// TwinCAT 3 PLC project TcDynCollectionsTest
// Title: TwinCAT Dynamic Collections Test
// Company: FisoThemes
// Author: Goodwill Mzumala
// Description: Test solution for the TcDynCollections Library
// ProgramVersion: 3.1.4023.0
// libraries:
//   Tc2_Standard, * (Beckhoff Automation GmbH)
//   Tc2_System, * (Beckhoff Automation GmbH)
//   Tc2_Utilities, * (Beckhoff Automation GmbH)
//   Tc3_Module, * (Beckhoff Automation GmbH)
//   TcUnit, * (www.tcunit.org)
//   TwinCat Dynamic Collections, * (FisoThemes)
// project tree:
//   / PlcTask.TcTTO
//   POUs/Function Blocks/ FB_Array_List_Test_Suite.TcPOU, FB_Array_Test_Suite.TcPOU, FB_Ordered_Hash_Map_Test_Suite.TcPOU, FB_Ordered_Hash_Set_Test_Suite.TcPOU, FB_List_Test_Suite.TcPOU, FB_Queue_Test_Suite.TcPOU, FB_Deque_Test_Suite.TcPOU, FB_Stack_Test_Suite.TcPOU, FB_Tree_Map_Test_Suite.TcPOU, FB_Hash_Map_Test_Suite.TcPOU, FB_Tree_Set_Test_Suite.TcPOU, FB_Tree_Multiset_Test_Suite.TcPOU, FB_Hash_Set_Test_Suite.TcPOU
//   POUs/ MAIN.TcPOU
// (motion and I/O tree: see PLC project tcdyncollections)
// real-time tasks:
//   TASK PlcTask: cycle T#10ms, priority 20, ADS port 350
//   TASK PlcTestTask: cycle T#10ms, priority 21, ADS port 353

CONFIGURATION TcDynCollectionsTest
    RESOURCE PLC ON TwinCAT3
        TASK PlcTask(INTERVAL := T#10ms, PRIORITY := 20);
        PROGRAM MAIN WITH PlcTask : MAIN;
    END_RESOURCE
END_CONFIGURATION

// ---- POUs/MAIN.TcPOU
PROGRAM MAIN
VAR
	fbArray_List_Test_Suite : FB_Array_List_Test_Suite;
	fbList_Test_Suite : FB_List_Test_Suite;
	fbArray_Test_Suite : FB_Array_Test_Suite;
	fbQueue_Test_Suite : FB_Queue_Test_Suite;
	fbStack_Test_Suite : FB_Stack_Test_Suite;
	fbDeque_Test_Suite : FB_Deque_Test_Suite;
	fbTree_Set_Test_Suite : FB_Tree_Set_Test_Suite;
	fbTree_Map_Test_Suite : FB_Tree_Map_Test_Suite;
	fbTree_Multiset_Test_Suite : FB_Tree_Multiset_Test_Suite;
	fbHash_Set_Test_Suite : FB_Hash_Set_Test_Suite;
	fbHash_Map_Test_Suite : FB_Hash_Map_Test_Suite;
	fbOrdered_Hash_Set_Test_Suite : FB_Ordered_Hash_Set_Test_Suite;
	fbOrdered_Hash_Map_Test_Suite : FB_Ordered_Hash_Map_Test_Suite;
END_VAR

TcUnit.RUN();

END_PROGRAM

// ---- POUs/Function Blocks/FB_Array_List_Test_Suite.TcPOU
FUNCTION_BLOCK FB_Array_List_Test_Suite EXTENDS TcUnit.FB_TestSuite
VAR
END_VAR

THIS^.Append_Items_And_Check_If_Count_Changes();
THIS^.Append_Items_And_Get_Items();
THIS^.Prepend_Items_And_Get_Items();
THIS^.Append_Items_Reverse_The_List_And_Get_Items();
THIS^.Append_Find_Item_Indices_And_Get_Items_With_Them();
THIS^.Remove_Tests();
THIS^.Set_Value_At_Index_To_Item_And_Get_Item();

// Test appending multiple elements, finds them and verify values using the get method.
METHOD Append_Find_Item_Indices_And_Get_Items_With_Them
VAR_INST
	fbList 		: TcDynCollections.FB_Array_List(0);
	Idx 		: ARRAY[0..4] OF TcDynCollections.T_Position;
	arbValue 	: ARRAY[0..2] OF BOOL := [TRUE, TRUE];
	arnValue 	: ARRAY[0..2] OF INT := [33, 33];
	arsValue 	: ARRAY[0..2] OF STRING := ['I love cats.', 'I love cats.'];
	arwsValue 	: ARRAY[0..2] OF WSTRING := ["I love dogs.", "I love dogs."];
	arfValue 	: ARRAY[0..2] OF LREAL := [21.3, 21.3];
END_VAR
TcUnit.TEST('Append_Find_Item_Indices_And_Get_Items_With_Them');

	fbList
		.Append(arbValue[0])
		.Append(arnValue[0])
		.Append(arsValue[0])
		.Append(arwsValue[0])
		.Append(arfValue[0]);

	// Make the strings dirty. 	
	arsValue[0] 	:= 'kjhsadkfjvhbkjhdfbkvsjhbfkvjhsbkfv';
	arwsValue[0] 	:= "kjhsadkfjvhbkjhdfbkvsjhbfkvjhsbkfv";
	arsValue[0] 	:= 'I love cats.';
	arwsValue[0] 	:= "I love dogs.";
		
	fbList
		.Search(arbValue[0], Index => Idx[0])
		.Search(arnValue[0], Index => Idx[1])
		.Search(arsValue[0], Index => Idx[2])
		.Search(arwsValue[0],Index => Idx[3])
		.Search(arfValue[0], Index => Idx[4]);
		
	fbList
		.Get(Idx[0], arbValue[2])
		.Get(Idx[1], arnValue[2])
		.Get(Idx[2], arsValue[2])
		.Get(Idx[3], arwsValue[2])
		.Get(Idx[4], arfValue[2]);
		
	THIS^.AssertEquals_DINT(5, fbList._Count, 'List item count must be 5 after after appending items to list.');
	THIS^.AssertEquals_BOOL(arbValue[1], arbValue[2], 'Appended BOOL item is not what is expected after the get operation.');
	THIS^.AssertEquals_INT(arnValue[1], arnValue[2], 'Appended INT item is not what is expected after the get operation.');
	THIS^.AssertEquals_STRING(arsValue[1], arsValue[2], 'Appended STRING item is not what is expected after the get operation.');
	THIS^.AssertEquals_WSTRING(arwsValue[1], arwsValue[2], 'Appended STRING item is not what is expected after the get operation.');
	THIS^.AssertEquals_LREAL(arfValue[1], arfValue[2],0.01, 'Appended LREAL item is not what is expected after the get operation.');

	TEST_FINISHED();
END_METHOD

// 1) Test that a newly created FB_Array_List has an item count of 0 and is empty.
// 2) Test that after appending elements, the size increases accordingly and is no longer empty.
// 3) Test that after removing all elements, the size becomes 0 again and the list is empty.
METHOD Append_Items_And_Check_If_Count_Changes
VAR_INST
	fbList : TcDynCollections.FB_Array_List(0);
	nValue : INT := 33;
	sValue : STRING := 'I love cats.';
END_VAR
TcUnit.TEST('Append_Items_And_Check_If_Count_Changes');

	THIS^.AssertEquals_DINT(0, fbList._Count, 'List item count must be 0.');
	THIS^.AssertEquals_BOOL(TRUE, fbList._Empty, '_Empty property didnt return TRUE.');
	
	fbList
		.Append(nValue)
		.Append(sValue);
	
	THIS^.AssertEquals_DINT(2, fbList._Count, 'List item count must be 2 after appending values.');
	THIS^.AssertEquals_BOOL(FALSE, fbList._Empty, '_Empty property didnt return FALSE after appending value.');
	
	fbList.Clear();
	
	THIS^.AssertEquals_DINT(0, fbList._Count, 'List item count must be 0 after clearing list.');
	THIS^.AssertEquals_BOOL(TRUE, fbList._Empty, '_Empty property didnt return TRUE after clearing list.');
	
	TEST_FINISHED();
END_METHOD

// Test appending multiple elements and verify their order and values using the get method.
METHOD Append_Items_And_Get_Items
VAR_INST
	fbList 		: TcDynCollections.FB_Array_List(0);
	
	arbValue 	: ARRAY[0..2] OF BOOL := [TRUE, TRUE];
	arnValue 	: ARRAY[0..2] OF INT := [33, 33];
	arsValue 	: ARRAY[0..2] OF STRING := ['I love cats.', 'I love cats.'];
	arwsValue 	: ARRAY[0..2] OF WSTRING := ["I love dogs.", "I love dogs."];
	arfValue 	: ARRAY[0..2] OF LREAL := [21.3, 21.3];
END_VAR
TcUnit.TEST('Append_Items_And_Get_Items');

	fbList
		.Append(arbValue[0])
		.Append(arnValue[0])
		.Append(arsValue[0])
		.Append(arwsValue[0])
		.Append(arfValue[0]);
		
	fbList
		.Get(0, arbValue[2])
		.Get(1, arnValue[2])
		.Get(2, arsValue[2])
		.Get(3, arwsValue[2])
		.Get(4, arfValue[2]);
		
	THIS^.AssertEquals_DINT(5, fbList._Count, 'List item count must be 5 after after appending items to list.');
	THIS^.AssertEquals_BOOL(arbValue[1], arbValue[2], 'Appended BOOL item is not what is expected after the get operation.');
	THIS^.AssertEquals_INT(arnValue[1], arnValue[2], 'Appended INT item is not what is expected after the get operation.');
	THIS^.AssertEquals_STRING(arsValue[1], arsValue[2], 'Appended STRING item is not what is expected after the get operation.');
	THIS^.AssertEquals_WSTRING(arwsValue[1], arwsValue[2], 'Appended STRING item is not what is expected after the get operation.');
	THIS^.AssertEquals_LREAL(arfValue[1], arfValue[2],0.01, 'Appended LREAL item is not what is expected after the get operation.');

	TEST_FINISHED();
END_METHOD

// Test appending multiple elements, reversing their order and verifiying their order and values using the get method.
METHOD Append_Items_Reverse_The_List_And_Get_Items
VAR_INST
	fbList 		: TcDynCollections.FB_Array_List(0);
	
	arbValue 	: ARRAY[0..2] OF BOOL := [TRUE, TRUE];
	arnValue 	: ARRAY[0..2] OF INT := [33, 33];
	arsValue 	: ARRAY[0..2] OF STRING := ['I love cats.', 'I love cats.'];
	arwsValue 	: ARRAY[0..2] OF WSTRING := ["I love dogs.", "I love dogs."];
	arfValue 	: ARRAY[0..2] OF LREAL := [21.3, 21.3];
END_VAR
TcUnit.TEST('Append_Items_Reverse_The_List_And_Get_Items');

	fbList
		.Append(arbValue[0])
		.Append(arnValue[0])
		.Append(arsValue[0])
		.Append(arwsValue[0])
		.Append(arfValue[0])
		.Reverse();
		
	fbList
		.Get(4, arbValue[2])
		.Get(3, arnValue[2])
		.Get(2, arsValue[2])
		.Get(1, arwsValue[2])
		.Get(0, arfValue[2]);
		
	THIS^.AssertEquals_DINT(5, fbList._Count, 'List item count must be 5 after after appending items to list.');
	THIS^.AssertEquals_BOOL(arbValue[1], arbValue[2], 'Appended BOOL item is not what is expected after the get operation.');
	THIS^.AssertEquals_INT(arnValue[1], arnValue[2], 'Appended INT item is not what is expected after the get operation.');
	THIS^.AssertEquals_STRING(arsValue[1], arsValue[2], 'Appended STRING item is not what is expected after the get operation.');
	THIS^.AssertEquals_WSTRING(arwsValue[1], arwsValue[2], 'Appended STRING item is not what is expected after the get operation.');
	THIS^.AssertEquals_LREAL(arfValue[1], arfValue[2],0.01, 'Appended LREAL item is not what is expected after the get operation.');

	TEST_FINISHED();
END_METHOD

// Test prepending multiple elements and verify their order and values using the get method.
METHOD Prepend_Items_And_Get_Items
VAR_INST
	fbList 		: TcDynCollections.FB_Array_List(0);
	
	arbValue 	: ARRAY[0..2] OF BOOL := [TRUE, TRUE];
	arnValue 	: ARRAY[0..2] OF INT := [33, 33];
	arsValue 	: ARRAY[0..2] OF STRING := ['I love cats.', 'I love cats.'];
	arwsValue 	: ARRAY[0..2] OF WSTRING := ["I love dogs.", "I love dogs."];
	arfValue 	: ARRAY[0..2] OF LREAL := [21.3, 21.3];
END_VAR
TcUnit.TEST('Prepend_Items_And_Get_Items');

	fbList
		.Prepend(arbValue[0])
		.Prepend(arnValue[0])
		.Prepend(arsValue[0])
		.Prepend(arwsValue[0])
		.Prepend(arfValue[0]);
		
	fbList
		.Get(4, arbValue[2])
		.Get(3, arnValue[2])
		.Get(2, arsValue[2])
		.Get(1, arwsValue[2])
		.Get(0, arfValue[2]);
		
	THIS^.AssertEquals_DINT(5, fbList._Count, 'List item count must be 5 after after appending items to list.');
	THIS^.AssertEquals_BOOL(arbValue[1], arbValue[2], 'Appended BOOL item is not what is expected after the get operation.');
	THIS^.AssertEquals_INT(arnValue[1], arnValue[2], 'Appended INT item is not what is expected after the get operation.');
	THIS^.AssertEquals_STRING(arsValue[1], arsValue[2], 'Appended STRING item is not what is expected after the get operation.');
	THIS^.AssertEquals_WSTRING(arwsValue[1], arwsValue[2], 'Appended STRING item is not what is expected after the get operation.');
	THIS^.AssertEquals_LREAL(arfValue[1], arfValue[2],0.01, 'Appended LREAL item is not what is expected after the get operation.');

	TEST_FINISHED();
END_METHOD

// Test appending multiple elements, removing first item, verifying the size and values.
// 
METHOD Remove_Tests
VAR_INST
	fbList 		: TcDynCollections.FB_Array_List(0);
	i 			: TcDynCollections.T_Position;
	n 			: TcDynCollections.T_Capacity;
	arbValue 	: ARRAY[0..2] OF BOOL := [TRUE, TRUE];
	arnValue 	: ARRAY[0..2] OF INT := [33, 33];
	arsValue 	: ARRAY[0..2] OF STRING := ['I love cats.', 'I love cats.'];
	arwsValue 	: ARRAY[0..2] OF WSTRING := ["I love dogs.", "I love dogs."];
	arfValue 	: ARRAY[0..2] OF LREAL := [21.3, 21.3];
END_VAR
TcUnit.TEST('Remove_Tests');

	fbList
		.Append(arbValue[0])
		.Append(arnValue[0])
		.Append(arsValue[0])
		.Append(arwsValue[0])
		.Append(arfValue[0]);
		
	fbList
		.Remove(arbValue[0])
		.Get(0, arnValue[2]);
		
	THIS^.AssertEquals_DINT(4, fbList._Count, 'List item count must be 4 after appending and removing fisrt item at from the list.');
	THIS^.AssertEquals_INT(arnValue[1], arnValue[2],'');
	
	fbList
		.Prepend(arbValue[0])
		.Remove_At(2)
		.Get(2, arwsValue[2]);
		
	THIS^.AssertEquals_DINT(4, fbList._Count, 'List item count must be 4 after prepending removed item and removing item in index 2 of the list.');
	THIS^.AssertEquals_WSTRING(arwsValue[1], arwsValue[2], '');
	
	fbList
		.Insert(2, arsValue[0])
		.Remove_Last()
		.Get(3, arwsValue[2]);
		
	THIS^.AssertEquals_DINT(4, fbList._Count, 'List item count must be 4 after inserting removed from index 2 item and removing the last item in the list.');
	THIS^.AssertEquals_WSTRING(arwsValue[1], arwsValue[2], '');
	
	n := fbList._Count;
	FOR i := 0 TO n - 1 DO
		fbList.Remove_Last();
		END_FOR
		
	THIS^.AssertEquals_DINT(0, fbList._Count, 'List item count must be zero after removing all items from the back.');
	THIS^.AssertEquals_BOOL(TRUE, fbList._Empty, 'List _Empty property must be zero TRUE removing all items from the back.');
	
	FOR i := 0 TO 4 DO fbList.Prepend(arwsValue); END_FOR
	
	THIS^.AssertEquals_DINT(5, fbList._Count, 'Failed to prepend items to list for checking removing all items from the front.');
	
	n := fbList._Count;
	FOR i := 0 TO n - 1 DO
		fbList.Remove_At(0);
		END_FOR
		
	THIS^.AssertEquals_DINT(0, fbList._Count, 'List item count must be zero after removing all items from the front.');
	THIS^.AssertEquals_BOOL(TRUE, fbList._Empty, 'List _Empty property must be zero TRUE removing all items from the front.');

	TEST_FINISHED();
END_METHOD

// Test appending multiple elements and verify their order and values using the get method.
METHOD Set_Value_At_Index_To_Item_And_Get_Item
VAR_INST
	fbList 		: TcDynCollections.FB_Array_List(5);
	
	arbValue 	: ARRAY[0..2] OF BOOL := [TRUE, TRUE];
	arnValue 	: ARRAY[0..2] OF INT := [33, 33];
	arsValue 	: ARRAY[0..2] OF STRING := ['I love cats.', 'I love cats.'];
	arwsValue 	: ARRAY[0..2] OF WSTRING := ["I love dogs.", "I love dogs."];
	arfValue 	: ARRAY[0..2] OF LREAL := [21.3, 21.3];
END_VAR
TcUnit.TEST('Set_Value_At_Index_To_Item_And_Get_Item');

	fbList
		.Set(0, arbValue[0])
		.Set(1, arnValue[0])
		.Set(2, arsValue[0])
		.Set(3, arwsValue[0])
		.Set(4, arfValue[0]);
		
	fbList
		.Get(0, arbValue[2])
		.Get(1, arnValue[2])
		.Get(2, arsValue[2])
		.Get(3, arwsValue[2])
		.Get(4, arfValue[2]);
		
	THIS^.AssertEquals_DINT(5, fbList._Count, 'List item count must be 5 after after appending items to list.');
	THIS^.AssertEquals_BOOL(arbValue[1], arbValue[2], 'Appended BOOL item is not what is expected after the get operation.');
	THIS^.AssertEquals_INT(arnValue[1], arnValue[2], 'Appended INT item is not what is expected after the get operation.');
	THIS^.AssertEquals_STRING(arsValue[1], arsValue[2], 'Appended STRING item is not what is expected after the get operation.');
	THIS^.AssertEquals_WSTRING(arwsValue[1], arwsValue[2], 'Appended STRING item is not what is expected after the get operation.');
	THIS^.AssertEquals_LREAL(arfValue[1], arfValue[2],0.01, 'Appended LREAL item is not what is expected after the get operation.');

	TEST_FINISHED();
END_METHOD

END_FUNCTION_BLOCK

// ---- POUs/Function Blocks/FB_List_Test_Suite.TcPOU
FUNCTION_BLOCK FB_List_Test_Suite EXTENDS TcUnit.FB_TestSuite
VAR
END_VAR

THIS^.Append_Items_And_Check_If_Count_Changes();
THIS^.Append_Items_And_Get_Items();
THIS^.Prepend_Items_And_Get_Items();
THIS^.Append_Items_Reverse_The_List_And_Get_Items();
THIS^.Append_Find_Item_Indices_And_Get_Items_With_Them();
THIS^.Remove_Tests();
THIS^.Set_Value_At_Index_To_Item_And_Get_Item();

// Test appending multiple elements, finds them and verify values using the get method.
METHOD Append_Find_Item_Indices_And_Get_Items_With_Them
VAR_INST
	fbList 		: TcDynCollections.FB_List;
	Idx 		: ARRAY[0..4] OF TcDynCollections.T_Position;
	arbValue 	: ARRAY[0..2] OF BOOL := [TRUE, TRUE];
	arnValue 	: ARRAY[0..2] OF INT := [33, 33];
	arsValue 	: ARRAY[0..2] OF STRING := ['I love cats.', 'I love cats.'];
	arwsValue 	: ARRAY[0..2] OF WSTRING := ["I love dogs.", "I love dogs."];
	arfValue 	: ARRAY[0..2] OF LREAL := [21.3, 21.3];
END_VAR
TcUnit.TEST('Append_Find_Item_Indices_And_Get_Items_With_Them');

	fbList
		.Append(arbValue[0])
		.Append(arnValue[0])
		.Append(arsValue[0])
		.Append(arwsValue[0])
		.Append(arfValue[0]);

	// Make the strings dirty. 	
	arsValue[0] 	:= 'kjhsadkfjvhbkjhdfbkvsjhbfkvjhsbkfv';
	arwsValue[0] 	:= "kjhsadkfjvhbkjhdfbkvsjhbfkvjhsbkfv";
	arsValue[0] 	:= 'I love cats.';
	arwsValue[0] 	:= "I love dogs.";
		
	fbList
		.Search(arbValue[0], Index => Idx[0])
		.Search(arnValue[0], Index => Idx[1])
		.Search(arsValue[0], Index => Idx[2])
		.Search(arwsValue[0],Index => Idx[3])
		.Search(arfValue[0], Index => Idx[4]);
		
	fbList
		.Get(Idx[0], arbValue[2])
		.Get(Idx[1], arnValue[2])
		.Get(Idx[2], arsValue[2])
		.Get(Idx[3], arwsValue[2])
		.Get(Idx[4], arfValue[2]);
		
	THIS^.AssertEquals_DINT(5, fbList._Count, 'List item count must be 5 after after appending items to list.');
	THIS^.AssertEquals_BOOL(arbValue[1], arbValue[2], 'Appended BOOL item is not what is expected after the get operation.');
	THIS^.AssertEquals_INT(arnValue[1], arnValue[2], 'Appended INT item is not what is expected after the get operation.');
	THIS^.AssertEquals_STRING(arsValue[1], arsValue[2], 'Appended STRING item is not what is expected after the get operation.');
	THIS^.AssertEquals_WSTRING(arwsValue[1], arwsValue[2], 'Appended STRING item is not what is expected after the get operation.');
	THIS^.AssertEquals_LREAL(arfValue[1], arfValue[2],0.01, 'Appended LREAL item is not what is expected after the get operation.');

	TEST_FINISHED();
END_METHOD

// 1) Test that a newly created FB_Array_List has an item count of 0 and is empty.
// 2) Test that after appending elements, the size increases accordingly and is no longer empty.
// 3) Test that after removing all elements, the size becomes 0 again and the list is empty.
METHOD Append_Items_And_Check_If_Count_Changes
VAR_INST
	fbList : TcDynCollections.FB_List;
	nValue : INT := 33;
	sValue : STRING := 'I love cats.';
END_VAR
TcUnit.TEST('Append_Items_And_Check_If_Count_Changes');

	THIS^.AssertEquals_DINT(0, fbList._Count, 'List item count must be 0.');
	THIS^.AssertEquals_BOOL(TRUE, fbList._Empty, 'Is_Empty property didnt return TRUE.');
	
	fbList
		.Append(nValue)
		.Append(sValue);
	
	THIS^.AssertEquals_DINT(2, fbList._Count, 'List item count must be 2 after appending values.');
	THIS^.AssertEquals_BOOL(FALSE, fbList._Empty, 'Is_Empty property didnt return FALSE after appending value.');
	
	fbList.Clear();
	
	THIS^.AssertEquals_DINT(0, fbList._Count, 'List item count must be 0 after clearing list.');
	THIS^.AssertEquals_BOOL(TRUE, fbList._Empty, 'Is_Empty property didnt return TRUE after clearing list.');
	
	TEST_FINISHED();
END_METHOD

// Test appending multiple elements and verify their order and values using the get method.
METHOD Append_Items_And_Get_Items
VAR_INST
	fbList 		: TcDynCollections.FB_List;
	
	arbValue 	: ARRAY[0..2] OF BOOL := [TRUE, TRUE];
	arnValue 	: ARRAY[0..2] OF INT := [33, 33];
	arsValue 	: ARRAY[0..2] OF STRING := ['I love cats.', 'I love cats.'];
	arwsValue 	: ARRAY[0..2] OF WSTRING := ["I love dogs.", "I love dogs."];
	arfValue 	: ARRAY[0..2] OF LREAL := [21.3, 21.3];
END_VAR
TcUnit.TEST('Append_Items_And_Get_Items');

	fbList
		.Append(arbValue[0])
		.Append(arnValue[0])
		.Append(arsValue[0])
		.Append(arwsValue[0])
		.Append(arfValue[0]);
		
	fbList
		.Get(0, arbValue[2])
		.Get(1, arnValue[2])
		.Get(2, arsValue[2])
		.Get(3, arwsValue[2])
		.Get(4, arfValue[2]);
		
	THIS^.AssertEquals_DINT(5, fbList._Count, 'List item count must be 5 after after appending items to list.');
	THIS^.AssertEquals_BOOL(arbValue[1], arbValue[2], 'Appended BOOL item is not what is expected after the get operation.');
	THIS^.AssertEquals_INT(arnValue[1], arnValue[2], 'Appended INT item is not what is expected after the get operation.');
	THIS^.AssertEquals_STRING(arsValue[1], arsValue[2], 'Appended STRING item is not what is expected after the get operation.');
	THIS^.AssertEquals_WSTRING(arwsValue[1], arwsValue[2], 'Appended STRING item is not what is expected after the get operation.');
	THIS^.AssertEquals_LREAL(arfValue[1], arfValue[2],0.01, 'Appended LREAL item is not what is expected after the get operation.');

	TEST_FINISHED();
END_METHOD

// Test appending multiple elements, reversing their order and verifiying their order and values using the get method.
METHOD Append_Items_Reverse_The_List_And_Get_Items
VAR_INST
	fbList 		: TcDynCollections.FB_List;
	
	arbValue 	: ARRAY[0..2] OF BOOL := [TRUE, TRUE];
	arnValue 	: ARRAY[0..2] OF INT := [33, 33];
	arsValue 	: ARRAY[0..2] OF STRING := ['I love cats.', 'I love cats.'];
	arwsValue 	: ARRAY[0..2] OF WSTRING := ["I love dogs.", "I love dogs."];
	arfValue 	: ARRAY[0..2] OF LREAL := [21.3, 21.3];
END_VAR
TcUnit.TEST('Append_Items_Reverse_The_List_And_Get_Items');

	fbList
		.Append(arbValue[0])
		.Append(arnValue[0])
		.Append(arsValue[0])
		.Append(arwsValue[0])
		.Append(arfValue[0])
		.Reverse();
		
	fbList
		.Get(4, arbValue[2])
		.Get(3, arnValue[2])
		.Get(2, arsValue[2])
		.Get(1, arwsValue[2])
		.Get(0, arfValue[2]);
		
	THIS^.AssertEquals_DINT(5, fbList._Count, 'List item count must be 5 after after appending items to list.');
	THIS^.AssertEquals_BOOL(arbValue[1], arbValue[2], 'Appended BOOL item is not what is expected after the get operation.');
	THIS^.AssertEquals_INT(arnValue[1], arnValue[2], 'Appended INT item is not what is expected after the get operation.');
	THIS^.AssertEquals_STRING(arsValue[1], arsValue[2], 'Appended STRING item is not what is expected after the get operation.');
	THIS^.AssertEquals_WSTRING(arwsValue[1], arwsValue[2], 'Appended STRING item is not what is expected after the get operation.');
	THIS^.AssertEquals_LREAL(arfValue[1], arfValue[2],0.01, 'Appended LREAL item is not what is expected after the get operation.');

	TEST_FINISHED();
END_METHOD

// Test prepending multiple elements and verify their order and values using the get method.
METHOD Prepend_Items_And_Get_Items
VAR_INST
	fbList 		: TcDynCollections.FB_List;
	arsPrint 	: ARRAY[0..4] OF STRING;
	arbValue 	: ARRAY[0..2] OF BOOL := [TRUE, TRUE];
	arnValue 	: ARRAY[0..2] OF INT := [33, 33];
	arsValue 	: ARRAY[0..2] OF STRING := ['I love cats.', 'I love cats.'];
	arwsValue 	: ARRAY[0..2] OF WSTRING := ["I love dogs.", "I love dogs."];
	arfValue 	: ARRAY[0..2] OF LREAL := [21.3, 21.3];
END_VAR
TcUnit.TEST('Prepend_Items_And_Get_Items');

	fbList
		.Prepend(arbValue[0])
		.Prepend(arnValue[0])
		.Prepend(arsValue[0])
		.Prepend(arwsValue[0])
		.Prepend(arfValue[0]);
		
	fbList
		.Get(4, arbValue[2])
		.Get(3, arnValue[2])
		.Get(2, arsValue[2])
		.Get(1, arwsValue[2])
		.Get(0, arfValue[2]);
		
	THIS^.AssertEquals_DINT(5, fbList._Count, 'List item count must be 5 after after appending items to list.');
	THIS^.AssertEquals_BOOL(arbValue[1], arbValue[2], 'Appended BOOL item is not what is expected after the get operation.');
	THIS^.AssertEquals_INT(arnValue[1], arnValue[2], 'Appended INT item is not what is expected after the get operation.');
	THIS^.AssertEquals_STRING(arsValue[1], arsValue[2], 'Appended STRING item is not what is expected after the get operation.');
	THIS^.AssertEquals_WSTRING(arwsValue[1], arwsValue[2], 'Appended STRING item is not what is expected after the get operation.');
	THIS^.AssertEquals_LREAL(arfValue[1], arfValue[2],0.01, 'Appended LREAL item is not what is expected after the get operation.');

	TEST_FINISHED();
END_METHOD

// Test appending multiple elements, removing first item, verifying the size and values.
METHOD Remove_Tests
VAR_INST
	fbList 		: TcDynCollections.FB_List;
	i 			: TcDynCollections.T_Position;
	n 			: TcDynCollections.T_Capacity;
	arbValue 	: ARRAY[0..2] OF BOOL := [TRUE, TRUE];
	arnValue 	: ARRAY[0..2] OF INT := [33, 33];
	arsValue 	: ARRAY[0..2] OF STRING := ['I love cats.', 'I love cats.'];
	arwsValue 	: ARRAY[0..2] OF WSTRING := ["I love dogs.", "I love dogs."];
	arfValue 	: ARRAY[0..2] OF LREAL := [21.3, 21.3];
END_VAR
TcUnit.TEST('Remove_Tests');

	fbList
		.Append(arbValue[0])
		.Append(arnValue[0])
		.Append(arsValue[0])
		.Append(arwsValue[0])
		.Append(arfValue[0]);
		
	fbList
		.Remove(arbValue[0])
		.Get(0, arnValue[2]);
		
	THIS^.AssertEquals_DINT(4, fbList._Count, 'List item count must be 4 after appending and removing fisrt item at from the list.');
	THIS^.AssertEquals_INT(arnValue[1], arnValue[2],'');
	
	fbList
		.Prepend(arbValue[0])
		.Remove_At(2)
		.Get(2, arwsValue[2]);
		
	THIS^.AssertEquals_DINT(4, fbList._Count, 'List item count must be 4 after prepending removed item and removing item in index 2 of the list.');
	THIS^.AssertEquals_WSTRING(arwsValue[1], arwsValue[2], '');
	
	fbList
		.Insert(2, arsValue[0])
		.Remove_At(fbList._Count - 1)
		.Get(3, arwsValue[2]);
		
	THIS^.AssertEquals_DINT(4, fbList._Count, 'List item count must be 4 after inserting removed from index 2 item and removing the last item in the list.');
	THIS^.AssertEquals_WSTRING(arwsValue[1], arwsValue[2], '');

	n := fbList._Count;
	FOR i := 0 TO n DO
		fbList.Remove_At(fbList._Count - 1);
		END_FOR
		
	THIS^.AssertEquals_DINT(0, fbList._Count, 'List item count must be zero after removing all items from the back.');
	THIS^.AssertEquals_BOOL(TRUE, fbList._Empty, 'List Is_Empty property must be zero TRUE removing all items from the back.');

	FOR i := 0 TO 4 DO fbList.Prepend(arwsValue); END_FOR
	
	THIS^.AssertEquals_DINT(5, fbList._Count, 'Failed to prepend items to list for checking removing all items from the front.');
	
	n := fbList._Count;
	FOR i := 0 TO n - 1 DO
		fbList.Remove_At(0);
		END_FOR
		
	THIS^.AssertEquals_DINT(0, fbList._Count, 'List item count must be zero after removing all items from the front.');
	THIS^.AssertEquals_BOOL(TRUE, fbList._Empty, 'List Is_Empty property must be zero TRUE removing all items from the front.');

	TEST_FINISHED();
END_METHOD

// Test appending multiple elements and verify their order and values using the get method.
METHOD Set_Value_At_Index_To_Item_And_Get_Item
VAR_INST
	fbList 		: TcDynCollections.FB_List;
	
	arbValue 	: ARRAY[0..2] OF BOOL := [TRUE, TRUE];
	arnValue 	: ARRAY[0..2] OF INT := [33, 33];
	arsValue 	: ARRAY[0..2] OF STRING := ['I love cats.', 'I love cats.'];
	arwsValue 	: ARRAY[0..2] OF WSTRING := ["I love dogs.", "I love dogs."];
	arfValue 	: ARRAY[0..2] OF LREAL := [21.3, 21.3];
END_VAR
TcUnit.TEST('Set_Value_At_Index_To_Item_And_Get_Item');

	fbList
		.Resize(5)
		.Set(0, arbValue[0])
		.Set(1, arnValue[0])
		.Set(2, arsValue[0])
		.Set(3, arwsValue[0])
		.Set(4, arfValue[0]);
		
	fbList
		.Get(0, arbValue[2])
		.Get(1, arnValue[2])
		.Get(2, arsValue[2])
		.Get(3, arwsValue[2])
		.Get(4, arfValue[2]);
		
	THIS^.AssertEquals_DINT(5, fbList._Count, 'List item count must be 5 after after appending items to list.');
	THIS^.AssertEquals_BOOL(arbValue[1], arbValue[2], 'Get BOOL item is not what is expected after the get operation.');
	THIS^.AssertEquals_INT(arnValue[1], arnValue[2], 'Get INT item is not what is expected after the get operation.');
	THIS^.AssertEquals_STRING(arsValue[1], arsValue[2], 'Get STRING item is not what is expected after the get operation.');
	THIS^.AssertEquals_WSTRING(arwsValue[1], arwsValue[2], 'Get STRING item is not what is expected after the get operation.');
	THIS^.AssertEquals_LREAL(arfValue[1], arfValue[2],0.01, 'Get LREAL item is not what is expected after the get operation.');

	TEST_FINISHED();
END_METHOD

END_FUNCTION_BLOCK

// ---- POUs/Function Blocks/FB_Array_Test_Suite.TcPOU
FUNCTION_BLOCK FB_Array_Test_Suite EXTENDS TcUnit.FB_TestSuite
VAR
END_VAR

Create_Empty_Array_And_Array_With_Item_And_Check_Count();
Set_Value_At_Index_To_Item_And_Get_Item();
Set_Items_Reverse_The_Array_And_Get_Items();
Set_And_Find_Item_Indices_Then_Get_Items();

// 1) Test that a newly created FB_Array_List has an item count of 0 and is empty.
// 2) Test that after appending elements, the size increases accordingly and is no longer empty.
// 3) Test that after removing all elements, the size becomes 0 again and the list is empty.
METHOD Create_Empty_Array_And_Array_With_Item_And_Check_Count
VAR_INST
	fbEmpty_Array : TcDynCollections.FB_Array(0);
	fbArray : TcDynCollections.FB_Array(2);
END_VAR
TcUnit.TEST('Create_Empty_Array_And_Array_With_Item_And_Check_Count');

	THIS^.AssertEquals_DINT(0, fbEmpty_Array._Count, 'Array item count must be 0.');
	THIS^.AssertEquals_BOOL(TRUE, fbEmpty_Array._Empty, 'Array _Empty property didnt return TRUE.');
	
	THIS^.AssertEquals_DINT(2, fbArray._Count, 'Array item count must be 2.');
	THIS^.AssertEquals_BOOL(FALSE, fbArray._Empty, 'Array _Empty property didnt return FALSE after appending value.');
	
	TEST_FINISHED();
END_METHOD

// Test appending multiple elements, finds them and verify values using the get method.
METHOD Set_And_Find_Item_Indices_Then_Get_Items
VAR_INST
	fbArray 		: TcDynCollections.FB_Array(5);
	Idx 		: ARRAY[0..4] OF TcDynCollections.T_Position;
	arbValue 	: ARRAY[0..2] OF BOOL := [TRUE, TRUE];
	arnValue 	: ARRAY[0..2] OF INT := [33, 33];
	arsValue 	: ARRAY[0..2] OF STRING := ['I love cats.', 'I love cats.'];
	arwsValue 	: ARRAY[0..2] OF WSTRING := ["I love dogs.", "I love dogs."];
	arfValue 	: ARRAY[0..2] OF LREAL := [21.3, 21.3];
END_VAR
TcUnit.TEST('Set_And_Find_Item_Indices_Then_Get_Items');

	fbArray
		.Set(0, arbValue[0])
		.Set(1, arnValue[0])
		.Set(2, arsValue[0])
		.Set(3, arwsValue[0])
		.Set(4, arfValue[0]);

	// Make the strings dirty. 	
	arsValue[0] 	:= 'kjhsadkfjvhbkjhdfbkvsjhbfkvjhsbkfv';
	arwsValue[0] 	:= "kjhsadkfjvhbkjhdfbkvsjhbfkvjhsbkfv";
	arsValue[0] 	:= 'I love cats.';
	arwsValue[0] 	:= "I love dogs.";
		
	fbArray
		.Search(arbValue[0], Index => Idx[0])
		.Search(arnValue[0], Index => Idx[1])
		.Search(arsValue[0], Index => Idx[2])
		.Search(arwsValue[0],Index => Idx[3])
		.Search(arfValue[0], Index => Idx[4]);
		
	fbArray
		.Get(Idx[0], arbValue[2])
		.Get(Idx[1], arnValue[2])
		.Get(Idx[2], arsValue[2])
		.Get(Idx[3], arwsValue[2])
		.Get(Idx[4], arfValue[2]);
		
	THIS^.AssertEquals_DINT(5, fbArray._Count, 'Array item count must be 5 after after appending items to list.');
	THIS^.AssertEquals_BOOL(arbValue[1], arbValue[2], 'Set BOOL item is not what is expected after the get operation.');
	THIS^.AssertEquals_INT(arnValue[1], arnValue[2], 'Set INT item is not what is expected after the get operation.');
	THIS^.AssertEquals_STRING(arsValue[1], arsValue[2], 'Set STRING item is not what is expected after the get operation.');
	THIS^.AssertEquals_WSTRING(arwsValue[1], arwsValue[2], 'Set STRING item is not what is expected after the get operation.');
	THIS^.AssertEquals_LREAL(arfValue[1], arfValue[2],0.01, 'Set LREAL item is not what is expected after the get operation.');

	TEST_FINISHED();
END_METHOD

// Test appending multiple elements, reversing their order and verifiying their order and values using the get method.
METHOD Set_Items_Reverse_The_Array_And_Get_Items
VAR_INST
	fbArray 	: TcDynCollections.FB_Array(5);
	
	arbValue 	: ARRAY[0..2] OF BOOL := [TRUE, TRUE];
	arnValue 	: ARRAY[0..2] OF INT := [33, 33];
	arsValue 	: ARRAY[0..2] OF STRING := ['I love cats.', 'I love cats.'];
	arwsValue 	: ARRAY[0..2] OF WSTRING := ["I love dogs.", "I love dogs."];
	arfValue 	: ARRAY[0..2] OF LREAL := [21.3, 21.3];
END_VAR
TcUnit.TEST('Set_Items_Reverse_The_Array_And_Get_Items');

	fbArray
		.Set(0, arbValue[0])
		.Set(1, arnValue[0])
		.Set(2, arsValue[0])
		.Set(3, arwsValue[0])
		.Set(4, arfValue[0])
		.Reverse();
		
	fbArray
		.Get(4, arbValue[2])
		.Get(3, arnValue[2])
		.Get(2, arsValue[2])
		.Get(1, arwsValue[2])
		.Get(0, arfValue[2]);
		
	THIS^.AssertEquals_DINT(5, fbArray._Count, 'Array item count must be 5 after after appending items to list.');
	THIS^.AssertEquals_BOOL(arbValue[1], arbValue[2], 'Set BOOL item is not what is expected after the get operation.');
	THIS^.AssertEquals_INT(arnValue[1], arnValue[2], 'Set INT item is not what is expected after the get operation.');
	THIS^.AssertEquals_STRING(arsValue[1], arsValue[2], 'Set STRING item is not what is expected after the get operation.');
	THIS^.AssertEquals_WSTRING(arwsValue[1], arwsValue[2], 'Set STRING item is not what is expected after the get operation.');
	THIS^.AssertEquals_LREAL(arfValue[1], arfValue[2],0.01, 'Set LREAL item is not what is expected after the get operation.');

	TEST_FINISHED();
END_METHOD

// Test appending multiple elements and verify their order and values using the get method.
METHOD Set_Value_At_Index_To_Item_And_Get_Item
VAR_INST
	fbArray 	: TcDynCollections.FB_Array(5);
	
	arbValue 	: ARRAY[0..2] OF BOOL := [TRUE, TRUE];
	arnValue 	: ARRAY[0..2] OF INT := [33, 33];
	arsValue 	: ARRAY[0..2] OF STRING := ['I love cats.', 'I love cats.'];
	arwsValue 	: ARRAY[0..2] OF WSTRING := ["I love dogs.", "I love dogs."];
	arfValue 	: ARRAY[0..2] OF LREAL := [21.3, 21.3];
END_VAR
TcUnit.TEST('Set_Value_At_Index_To_Item_And_Get_Item');

	fbArray
		.Set(0, arbValue[0])
		.Set(1, arnValue[0])
		.Set(2, arsValue[0])
		.Set(3, arwsValue[0])
		.Set(4, arfValue[0]);
		
	fbArray
		.Get(0, arbValue[2])
		.Get(1, arnValue[2])
		.Get(2, arsValue[2])
		.Get(3, arwsValue[2])
		.Get(4, arfValue[2]);
		
	THIS^.AssertEquals_DINT(5, fbArray._Count, 'Array item count must be 5 after after appending items to list.');
	THIS^.AssertEquals_BOOL(arbValue[1], arbValue[2], 'Set BOOL item is not what is expected after the get operation.');
	THIS^.AssertEquals_INT(arnValue[1], arnValue[2], 'Set INT item is not what is expected after the get operation.');
	THIS^.AssertEquals_STRING(arsValue[1], arsValue[2], 'Set STRING item is not what is expected after the get operation.');
	THIS^.AssertEquals_WSTRING(arwsValue[1], arwsValue[2], 'Set STRING item is not what is expected after the get operation.');
	THIS^.AssertEquals_LREAL(arfValue[1], arfValue[2],0.01, 'Set LREAL item is not what is expected after the get operation.');

	TEST_FINISHED();
END_METHOD

END_FUNCTION_BLOCK

// ---- POUs/Function Blocks/FB_Queue_Test_Suite.TcPOU
FUNCTION_BLOCK FB_Queue_Test_Suite EXTENDS TcUnit.FB_TestSuite
VAR
END_VAR

Check_If_Clear_Empties_Items();
Check_If_Dequeue_Removes_First_Item();
Check_If_Enqueue_Adds_Items();
Check_If_Get_Returns_First_Item();
Check_If_Reverse_Reverses_Order_Of_Items();

METHOD Check_If_Clear_Empties_Items
VAR_INST
	fbQueue : FB_Queue;
	sItem : STRING := 'I love cats';
	nItem : INT := 42;
END_VAR
TcUnit.TEST('Check_If_Clear_Empties');
	fbQueue
		.Enqueue(sItem)
		.Enqueue(nItem)
		.Clear();
		
	THIS^.AssertEquals_DINT(0, fbQueue._Count, 'Queue was not empty after enqueueing data.');
	
	TEST_FINISHED();
END_METHOD

METHOD Check_If_Dequeue_Removes_First_Item
VAR_INST
	fbQueue : FB_Queue;
	sItem : STRING := 'I love cats';
	nItem : INT := 42;
END_VAR
TcUnit.TEST('Check_If_Dequeue_Removes_First_Item');
	fbQueue
		.Enqueue(sItem)
		.Enqueue(nItem)
		.Dequeue();
		
	THIS^.AssertEquals_DINT(1, fbQueue._Count, 'Queue failed to remove item.');
	
	TEST_FINISHED();
END_METHOD

METHOD Check_If_Enqueue_Adds_Items
VAR_INST
	fbQueue : FB_Queue;
	ipItems : I_Immutable_List;
	sItem : STRING := 'I love cats';
	nItem : INT := 42;
	sR_Item : STRING;
	nR_Item : INT;
END_VAR
TcUnit.TEST('Check_If_Enqueue_Adds_Items');
	
	fbQueue
		.Enqueue(sItem)
		.Enqueue_At_Front(nItem);
		
	ipItems := fbQueue._Values;
	
	ipItems
		.Get(0, nR_Item)
		.Get(1, sR_Item);
	
	THIS^.AssertEquals_DINT(2, fbQueue._Count, 'Queue item count is not accurate.');
	THIS^.AssertEquals_INT(42, nR_Item, 'Queue failed to enqueue int item correctly.');
	THIS^.AssertEquals_STRING('I love cats', sR_Item, 'Queue failed to enqueue string item correctly.');
	
	TEST_FINISHED();
END_METHOD

METHOD Check_If_Get_Returns_First_Item
VAR_INST
	fbQueue : FB_Queue;
	sItem : STRING := 'I love cats';
	nItem : INT := 42;
	sR_Item : STRING;
	nR_Item : INT;
END_VAR
TcUnit.TEST('Check_If_Get_Returns_First_Item');
	
	fbQueue
		.Enqueue(sItem)
		.Enqueue(nItem)
		.Get(sR_Item);
	
	THIS^.AssertEquals_STRING('I love cats', sR_Item, 'Queue failed to get first item enqueued (string) correctly.');
	
	TEST_FINISHED();
END_METHOD

METHOD Check_If_Reverse_Reverses_Order_Of_Items
VAR_INST
	fbQueue : FB_Queue;
	ipItems : I_Immutable_List;
	sItem : STRING := 'I love cats';
	nItem : INT := 42;
	sR_Item : STRING;
	nR_Item : INT;
END_VAR
TcUnit.TEST('Check_If_Reverse_Reverses_Order_Of_Items');
	
	fbQueue
		.Enqueue(sItem)
		.Enqueue(nItem)
		.Reverse();
		
	ipItems := fbQueue._Values;
	
	ipItems
		.Get(0, nR_Item)
		.Get(1, sR_Item);
	
	THIS^.AssertEquals_DINT(2, fbQueue._Count, 'Queue item count is not accurate.');
	THIS^.AssertEquals_INT(42, nR_Item, 'Queue failed to enqueue int item correctly.');
	THIS^.AssertEquals_STRING('I love cats', sR_Item, 'Queue failed to enqueue string item correctly.');
	
	TEST_FINISHED();
END_METHOD

END_FUNCTION_BLOCK

// ---- POUs/Function Blocks/FB_Stack_Test_Suite.TcPOU
FUNCTION_BLOCK FB_Stack_Test_Suite EXTENDS TcUnit.FB_TestSuite
VAR
END_VAR

Check_If_Clear_Empties_Items();
Check_If_Pop_Removes_Item();
Check_If_Push_Adds_Items();
Check_If_Get_Returns_Top_Item();
Check_If_Reverse_Reverses_Order_Of_Items();

METHOD Check_If_Clear_Empties_Items
VAR_INST
	fbStack : FB_Stack;
	sItem : STRING := 'I love cats';
	nItem : INT := 42;
END_VAR
TcUnit.TEST('Check_If_Clear_Empties');
	
	fbStack
		.Push(sItem)
		.Push(nItem)
		.Clear();
		
	THIS^.AssertEquals_DINT(0, fbStack._Count, 'Stack was not empty after pushing data.');
	
	TEST_FINISHED();
END_METHOD

METHOD Check_If_Get_Returns_Top_Item
VAR_INST
	fbStack : FB_Stack;
	ipItems : I_Immutable_List;
	sItem : STRING := 'I love cats';
	nItem : INT := 42;
	sR_Item : STRING;
	nR_Item : INT;
END_VAR
TcUnit.TEST('Check_If_Get_Returns_Top_Item');
	
	fbStack
		.Push(sItem)
		.Push(nItem)
		.Get(nR_Item);
	
	THIS^.AssertEquals_INT(42, nR_Item, 'Stack failed to get top item pushed (int) correctly.');
	
	TEST_FINISHED();
END_METHOD

METHOD Check_If_Pop_Removes_Item
VAR_INST
	fbStack : FB_Stack;
	sItem : STRING := 'I love cats';
	nItem : INT := 42;
END_VAR
TcUnit.TEST('Check_If_Pop_Removes_Item');
	
	fbStack
		.Push(sItem)
		.Push(nItem)
		.Pop();
		
	THIS^.AssertEquals_DINT(1, fbStack._Count, 'Stack failed to remove item.');
	
	TEST_FINISHED();
END_METHOD

METHOD Check_If_Push_Adds_Items
VAR_INST
	fbStack : FB_Stack;
	ipItems : I_Immutable_List;
	sItem : STRING := 'I love cats';
	nItem : INT := 42;
	sR_Item : STRING;
	nR_Item : INT;
END_VAR
TcUnit.TEST('Check_If_Push_Adds_Items');
	
	fbStack
		.Push(sItem)
		.Push(nItem);
		
	ipItems := fbStack._Values;
	
	ipItems
		.Get(0, nR_Item)
		.Get(1, sR_Item);
	
	THIS^.AssertEquals_DINT(2, fbStack._Count, 'Stack item count is not accurate.');
	THIS^.AssertEquals_INT(42, nR_Item, 'Stack failed to push int item correctly.');
	THIS^.AssertEquals_STRING('I love cats', sR_Item, 'Stack failed to push string item correctly.');
	
	TEST_FINISHED();
END_METHOD

METHOD Check_If_Reverse_Reverses_Order_Of_Items
VAR_INST
	fbStack : FB_Stack;
	ipItems : I_Immutable_List;
	sItem : STRING := 'I love cats';
	nItem : INT := 42;
	sR_Item : STRING;
	nR_Item : INT;
END_VAR
TcUnit.TEST('Check_If_Reverse_Reverses_Order_Of_Items');
	
	fbStack
		.Push(sItem)
		.Push(nItem)
		.Reverse();
		
	ipItems := fbStack._Values;
	
	ipItems
		.Get(0, sR_Item)
		.Get(1, nR_Item);
	
	THIS^.AssertEquals_DINT(2, fbStack._Count, 'Stack item count is not accurate.');
	THIS^.AssertEquals_INT(42, nR_Item, 'Stack failed to push int item correctly.');
	THIS^.AssertEquals_STRING('I love cats', sR_Item, 'Stack failed to push string item correctly.');
	
	TEST_FINISHED();
END_METHOD

END_FUNCTION_BLOCK

// ---- POUs/Function Blocks/FB_Deque_Test_Suite.TcPOU
FUNCTION_BLOCK FB_Deque_Test_Suite EXTENDS TcUnit.FB_TestSuite
VAR
END_VAR

Check_If_Clear_Empties_Items();
Check_If_Dequeue_At_Front_Removes_First_Item();
Check_If_Dequeue_At_Back_Removes_Last_Item();
Check_If_Enqueue_At_Back_Adds_Items();
Check_If_Enqueue_At_Front_Adds_Items();
Check_If_Back_Returns_Items_At_Back();
Check_If_Front_Returns_Items_At_Front();
Check_If_Reverse_Reverses_Order_Of_Items();

METHOD Check_If_Back_Returns_Items_At_Back
VAR_INST
	fbDeque : FB_Deque;
	sItem : STRING := 'I love cats';
	nItem : INT := 42;
	sR_Item : STRING;
	nR_Item : INT;
END_VAR
TcUnit.TEST('Check_If_Back_Returns_Items_At_Back');
	
	fbDeque
		.Enqueue_At_Back(sItem)
		.Enqueue_At_Back(nItem)
		.Back(nR_Item);
	
	THIS^.AssertEquals_INT(42, nR_Item, 'Deque failed to get item (int) at the back correctly.');
	
	TEST_FINISHED();
END_METHOD

METHOD Check_If_Clear_Empties_Items
VAR_INST
	fbDeque : FB_Deque;
	sItem : STRING := 'I love cats';
	nItem : INT := 42;
END_VAR
TcUnit.TEST('Check_If_Clear_Empties');
	
	fbDeque
		.Enqueue_At_Back (sItem)
		.Enqueue_At_Front(nItem)
		.Clear();
		
	THIS^.AssertEquals_DINT(0, fbDeque._Count, 'Deque was not empty after enqueueing data.');
	
	TEST_FINISHED();
END_METHOD

METHOD Check_If_Dequeue_At_Back_Removes_Last_Item
VAR_INST
	fbDeque : FB_Deque;
	sItem : STRING := 'I love cats';
	nItem : INT := 42;
	nR_Item : INT;
END_VAR
TcUnit.TEST('Check_If_Dequeue_At_Back_Removes_Last_Item');
	
	fbDeque
		.Enqueue_At_Front(sItem)
		.Enqueue_At_Front(nItem)
		.Dequeue_At_Back()
		._Values
			.Get(0, nR_Item);
		
	THIS^.AssertEquals_DINT(1, fbDeque._Count, 'Deque failed to remove item.');
	THIS^.AssertEquals_INT(42, nR_Item, 'Deque failed to get the last item.');
	
	TEST_FINISHED();
END_METHOD

METHOD Check_If_Dequeue_At_Front_Removes_First_Item
VAR_INST
	fbDeque : FB_Deque;
	sItem : STRING := 'I love cats';
	nItem : INT := 42;
	sR_Item : STRING;
END_VAR
TcUnit.TEST('Check_If_Dequeue_At_Front_Removes_First_Item');
	
	fbDeque
		.Enqueue_At_Front(sItem)
		.Enqueue_At_Front(nItem)
		.Dequeue_At_Front()
		._Values
			.Get(0, sR_Item);
		
	THIS^.AssertEquals_DINT(1, fbDeque._Count, 'Deque failed to remove item.');
	THIS^.AssertEquals_STRING('I love cats', sR_Item, 'Deque failed to get the first item.');
	
	TEST_FINISHED();
END_METHOD

METHOD Check_If_Enqueue_At_Back_Adds_Items
VAR_INST
	fbDeque : FB_Deque;
	ipItems : I_Immutable_List;
	sItem : STRING := 'I love cats';
	nItem : INT := 42;
	sR_Item : STRING;
	nR_Item : INT;
END_VAR
TcUnit.TEST('Check_If_Enqueue_At_Back_Adds_Items');

	fbDeque
		.Enqueue_At_Back(sItem)
		.Enqueue_At_Back(nItem);
		
	ipItems := fbDeque._Values;
	ipItems
		.Get(0, sR_Item)
		.Get(1, nR_Item);
	
	THIS^.AssertEquals_DINT(2, fbDeque._Count, 'Deque didnt enqueue elements at back corrrectly.');
	THIS^.AssertEquals_INT(42, nR_Item, 'Deque failed to get item (int) correctly.');
	THIS^.AssertEquals_STRING('I love cats', sR_Item, 'Deque failed to get item (string) correctly.');	
	
	TEST_FINISHED();
END_METHOD

METHOD Check_If_Enqueue_At_Front_Adds_Items
VAR_INST
	fbDeque : FB_Deque;
	ipItems : I_Immutable_List;
	sItem : STRING := 'I love cats';
	nItem : INT := 42;
	sR_Item : STRING;
	nR_Item : INT;
END_VAR
TcUnit.TEST('Check_If_Enqueue_At_Front_Adds_Items');

	fbDeque
		.Enqueue_At_Front(sItem)
		.Enqueue_At_Front(nItem);
		
	ipItems := fbDeque._Values;
	ipItems
		.Get(0, nR_Item)
		.Get(1, sR_Item);
	
	THIS^.AssertEquals_DINT(2, fbDeque._Count, 'Deque didnt enqueue elements at front corrrectly.');
	THIS^.AssertEquals_INT(42, nR_Item, 'Deque failed to get item (int) correctly.');
	THIS^.AssertEquals_STRING('I love cats', sR_Item, 'Deque failed to get item (string) correctly.');			
	
	TEST_FINISHED();
END_METHOD

METHOD Check_If_Front_Returns_Items_At_Front
VAR_INST
	fbDeque : FB_Deque;
	sItem : STRING := 'I love cats';
	nItem : INT := 42;
	sR_Item : STRING;
	nR_Item : INT;
END_VAR
TcUnit.TEST('Check_If_Front_Returns_Items_At_Front');
	
	fbDeque
		.Enqueue_At_Back(sItem)
		.Enqueue_At_Back(nItem)
		.Front(sR_Item);
	
	THIS^.AssertEquals_STRING('I love cats', sR_Item, 'Deque failed to get item (string) at the front correctly.');	
	
	TEST_FINISHED();
END_METHOD

METHOD Check_If_Reverse_Reverses_Order_Of_Items
VAR_INST
	fbDeque : FB_Deque;
	ipItems : I_Immutable_List;
	sItem : STRING := 'I love cats';
	nItem : INT := 42;
	sR_Item : STRING;
	nR_Item : INT;
END_VAR
TcUnit.TEST('Check_If_Reverse_Reverses_Order_Of_Items');

	fbDeque
		.Enqueue_At_Back(sItem)
		.Enqueue_At_Back(nItem)
		.Reverse();
		
	ipItems := fbDeque._Values;
	ipItems
		.Get(0, nR_Item)
		.Get(1, sR_Item);
	
	THIS^.AssertEquals_INT(42, nR_Item, 'Deque failed to get item (int) correctly.');
	THIS^.AssertEquals_STRING('I love cats', sR_Item, 'Deque failed to get item (string) correctly.');		
	
	TEST_FINISHED();
END_METHOD

END_FUNCTION_BLOCK

// ---- POUs/Function Blocks/FB_Tree_Set_Test_Suite.TcPOU
FUNCTION_BLOCK FB_Tree_Set_Test_Suite EXTENDS TcUnit.FB_TestSuite
VAR
END_VAR

Check_If_Clear_Empties_Items();
Check_If_Contains_Returns_True_If_Item_In_Set();
Check_If_Duplicate_Items_Cannot_Be_Inserted();
Check_If_Get_Values_Returns_Values_In_Specified_Order();
Check_If_Insert_Adds_Items();
Check_If_Remove_Removes_Items();
Check_If_Balanced_After_Removing_From_Left_Heavy_Tree();

METHOD Check_If_Balanced_After_Removing_From_Left_Heavy_Tree
VAR_INST
	fbSet : FB_Tree_Set;
	i, j : INT;
	arnItems : ARRAY[0..2] OF INT;
	ipItems : I_Immutable_List;
END_VAR
TcUnit.TEST('Check_If_Balanced_After_Removing_From_Left_Heavy_Tree');
	FOR i := 4 TO 1 BY -1 DO fbSet.Insert(i); END_FOR

	j := 3;
	fbSet._Traversal := T_BST_Traversal.Level_Order;
	ipItems := fbSet.Remove(j).Get_Values();

	ipItems
		.Get(0, arnItems[0])
		.Get(1, arnItems[1])
		.Get(2, arnItems[2]);
			
	THIS^.AssertEquals_DINT(3, fbSet._Count, 'Incorrect number of items retrieved after removing root item.');
	THIS^.AssertEquals_INT(2, arnItems[0], 'First value in level-order traversal is incorrect.');
	THIS^.AssertEquals_INT(1, arnItems[1], 'Second value in level-order traversal is incorrect.');
	THIS^.AssertEquals_INT(4, arnItems[2], 'Third value in level-order traversal is incorrect.');

TEST_FINISHED();
END_METHOD

METHOD Check_If_Clear_Empties_Items
VAR_INST
	fbSet : FB_Tree_Set;
	sItem : STRING := 'I love cats';
	nItem : INT := 42;
END_VAR
TcUnit.TEST('Check_If_Clear_Empties');
	fbSet
		.Insert(sItem)
		.Insert(nItem)
		.Clear();
		
	THIS^.AssertEquals_DINT(0, fbSet._Count, 'Set was not empty after inserting data.');
	
	TEST_FINISHED();
END_METHOD

METHOD Check_If_Contains_Returns_True_If_Item_In_Set
VAR_INST
	fbSet : FB_Tree_Set;
	sItem : STRING := 'I love cats';
	nItem : INT := 42;
	bResult : BOOL;
END_VAR
TcUnit.TEST('Check_If_Contains_Returns_True_If_Item_In_Set');

	bResult := fbSet
		.Insert(sItem)
		.Insert(nItem)
		.Contains(nItem);
		
	THIS^.AssertEquals_BOOL(TRUE, bResult, 'Failed to check if item is in set.');
	TEST_FINISHED();
END_METHOD

METHOD Check_If_Duplicate_Items_Cannot_Be_Inserted
VAR_INST
	fbSet : FB_Tree_Set;
	arnItems : ARRAY[0..5] OF DINT := [3,1,2,1,3,2];
	arnItems2 : ARRAY[0..2] OF DINT;
	ipItems : I_Immutable_List;
	i : DINT;
END_VAR
TcUnit.TEST('Check_If_Duplicate_Items_Cannot_Be_Inserted');

	FOR i := 0 TO 5 DO
    	fbSet.Insert(arnItems[i]);
    	END_FOR
		
	THIS^.AssertEquals_DINT(3, fbSet._Count, 'Set inserted duplicate items.');
	
	fbSet._Traversal := T_BST_Traversal.In_Order; // will get the values in ascending order

	ipItems := fbSet.Get_Values();
	ipItems
		.Get(0, arnItems2[0])
		.Get(1, arnItems2[1])
		.Get(2, arnItems2[2]);
		
	THIS^.AssertEquals_DINT(1, arnItems2[0],'');
	THIS^.AssertEquals_DINT(2, arnItems2[1],'');
	THIS^.AssertEquals_DINT(3, arnItems2[2],'');
		
	TEST_FINISHED();
END_METHOD

METHOD Check_If_Get_Values_Returns_Values_In_Specified_Order
VAR_INST
	fbSet : FB_Tree_Set;
	arnItems : ARRAY[0..3] OF DINT := [1,2,3,4];
	arnIn_Order, arnPre_Order, arnPost_Order, arnLevel_Order : ARRAY[0..3] OF DINT;
	i : DINT;
END_VAR
// Checked using: https://www.cs.usfca.edu/~galles/visualization/AVLtree.html
TcUnit.TEST('Check_If_Get_Values_Returns_Values_In_Specified_Order');

	FOR i := 0 TO 3 DO
    	fbSet.Insert(arnItems[i]);
    	END_FOR
		
	fbSet._Traversal := T_BST_Traversal.In_Order;
	fbSet.Get_Values()
		.Get(0, arnIn_Order[0])
		.Get(1, arnIn_Order[1]);
	fbSet.Get_Values()
		.Get(2, arnIn_Order[2])
		.Get(3, arnIn_Order[3]);
	THIS^.AssertEquals_DINT(1, arnIn_Order[0],'Failed to get item with in-order traversal.');
	THIS^.AssertEquals_DINT(2, arnIn_Order[1],'Failed to get item with in-order traversal.');
	THIS^.AssertEquals_DINT(3, arnIn_Order[2],'Failed to get item with in-order traversal.');
	THIS^.AssertEquals_DINT(4, arnIn_Order[3],'Failed to get item with in-order traversal.');
	
	fbSet._Traversal := T_BST_Traversal.Pre_Order;
	fbSet.Get_Values()
		.Get(0, arnPre_Order[0])
		.Get(1, arnPre_Order[1]);
	fbSet.Get_Values()
		.Get(2, arnPre_Order[2])
		.Get(3, arnPre_Order[3]);
	THIS^.AssertEquals_DINT(2, arnPre_Order[0],'Failed to get item with pre-order traversal.');
	THIS^.AssertEquals_DINT(1, arnPre_Order[1],'Failed to get item with pre-order traversal.');
	THIS^.AssertEquals_DINT(3, arnPre_Order[2],'Failed to get item with pre-order traversal.');
	THIS^.AssertEquals_DINT(4, arnPre_Order[3],'Failed to get item with pre-order traversal.');
	
	fbSet._Traversal := T_BST_Traversal.Post_Order; 
	fbSet.Get_Values()
		.Get(0, arnPost_Order[0])
		.Get(1, arnPost_Order[1]);
	fbSet.Get_Values()
		.Get(2, arnPost_Order[2])
		.Get(3, arnPost_Order[3]);
	THIS^.AssertEquals_DINT(1, arnPost_Order[0],'Failed to get item with post-order traversal.');
	THIS^.AssertEquals_DINT(4, arnPost_Order[1],'Failed to get item with post-order traversal.');
	THIS^.AssertEquals_DINT(3, arnPost_Order[2],'Failed to get item with post-order traversal.');
	THIS^.AssertEquals_DINT(2, arnPost_Order[3],'Failed to get item with post-order traversal.');
	
	fbSet._Traversal := T_BST_Traversal.Level_Order; // will get the values in ascending order
	fbSet.Get_Values()
		.Get(0, arnLevel_Order[0])
		.Get(1, arnLevel_Order[1]);
	fbSet.Get_Values()
		.Get(2, arnLevel_Order[2])
		.Get(3, arnLevel_Order[3]);
	THIS^.AssertEquals_DINT(2, arnLevel_Order[0],'Failed to get item with level-order traversal.');
	THIS^.AssertEquals_DINT(1, arnLevel_Order[1],'Failed to get item with level-order traversal.');
	THIS^.AssertEquals_DINT(3, arnLevel_Order[2],'Failed to get item with level-order traversal.');
	THIS^.AssertEquals_DINT(4, arnLevel_Order[3],'Failed to get item with level-order traversal.');
	
	TEST_FINISHED();
END_METHOD

METHOD Check_If_Insert_Adds_Items
VAR_INST
	fbSet : FB_Tree_Set;
	sItem : STRING := 'I love cats';
	nItem : INT := 42;
END_VAR
TcUnit.TEST('Check_If_Insert_Adds_Items');
	fbSet
		.Insert(sItem)
		.Insert(nItem);
		
	THIS^.AssertEquals_DINT(2, fbSet._Count, 'Failed to insert items into set.');
	
	TEST_FINISHED();
END_METHOD

METHOD Check_If_Remove_Removes_Items
VAR_INST
	fbSet : FB_Tree_Set;
	sItem : STRING := 'I love cats';
	nItem : INT := 42;
	fItem : LREAL := 37.4;
END_VAR
TcUnit.TEST('Check_If_Remove_Removes_Items');

	fbSet
		.Insert(sItem)
		.Insert(nItem)
		.Insert(fItem)
		.Remove(nItem);
		
	THIS^.AssertEquals_DINT(2, fbSet._Count, 'Failed to remove item in set.');
	THIS^.AssertEquals_BOOL(TRUE, fbSet.Contains(sItem), 'Failed to remove item in set.');
	THIS^.AssertEquals_BOOL(FALSE, fbSet.Contains(nItem), 'Failed to remove item in set.');
	THIS^.AssertEquals_BOOL(TRUE, fbSet.Contains(fItem), 'Failed to remove item in set.');	

	TEST_FINISHED();
END_METHOD

END_FUNCTION_BLOCK

// ---- POUs/Function Blocks/FB_Tree_Map_Test_Suite.TcPOU
FUNCTION_BLOCK FB_Tree_Map_Test_Suite EXTENDS TcUnit.FB_TestSuite
VAR
END_VAR

Check_If_Clear_Empties_Items();
Check_If_Insert_Adds_Items();
Check_If_Update_Updates_Items();
Check_If_Upsert_Updates_Items_Or_Adds_If_They_Dont_Exist();
Check_If_Remove_Removes_Items();
Check_If_Contains_Returns_True_If_Key_In_Map();
Check_If_Get_Key_Values_Returns_Keys_In_Specified_Order();
Check_If_Balanced_After_Removing_From_Left_Heavy_Tree();

METHOD Check_If_Balanced_After_Removing_From_Left_Heavy_Tree
VAR_INST
	fbMap : FB_Tree_Map;
	i, j : INT;
	arnKeys, arnValues : ARRAY[0..2] OF INT;
	ipKeys, ipValues : I_Immutable_List;
END_VAR
TcUnit.TEST('Check_If_Balanced_After_Removing_From_Left_Heavy_Tree');
	FOR i := 4 TO 1 BY -1 DO fbMap.Insert(i,i); END_FOR

	j := 3;
	fbMap._Traversal := T_BST_Traversal.Level_Order;
	ipKeys := fbMap.Remove(j).Get_Keys();
	ipValues := fbMap.Get_Values();
	
	ipKeys
		.Get(0, arnKeys[0])
		.Get(1, arnKeys[1])
		.Get(2, arnKeys[2]);

	ipValues
		.Get(0, arnValues[0])
		.Get(1, arnValues[1])
		.Get(2, arnValues[2]);
			
	THIS^.AssertEquals_DINT(3, fbMap._Count, 'Incorrect number of items retrieved after removing root item.');
	
	THIS^.AssertEquals_INT(2, arnKeys[0], 'First key in level-order traversal is incorrect.');
	THIS^.AssertEquals_INT(1, arnKeys[1], 'Second key in level-order traversal is incorrect.');
	THIS^.AssertEquals_INT(4, arnKeys[2], 'Third key in level-order traversal is incorrect.');
	
	THIS^.AssertEquals_INT(2, arnValues[0], 'First value in level-order traversal is incorrect.');
	THIS^.AssertEquals_INT(1, arnValues[1], 'Second value in level-order traversal is incorrect.');
	THIS^.AssertEquals_INT(4, arnValues[2], 'Third value in level-order traversal is incorrect.');

TEST_FINISHED();
END_METHOD

METHOD Check_If_Clear_Empties_Items
VAR_INST
	fbMap : FB_Tree_Map;
	sKey : STRING := 'I love cats';
	nValue : INT := 42;
END_VAR
TcUnit.TEST('Check_If_Clear_Empties');
	fbMap
		.Insert(sKey, nValue)
		.Clear();
		
	THIS^.AssertEquals_DINT(0, fbMap._Count, 'Map was not empty after inserting data.');
	
	TEST_FINISHED();
END_METHOD

METHOD Check_If_Contains_Returns_True_If_Key_In_Map
VAR_INST
	fbMap : FB_Tree_Map;
	sItem : STRING := 'I love cats';
	nItem : INT := 42;
	bResult : BOOL;
END_VAR
TcUnit.TEST('Check_If_Contains_Returns_True_If_Key_In_Map');

	bResult := fbMap
		.Insert(sItem, nItem)
		.Insert(nItem, sItem)
		.Contains(nItem);
		
	THIS^.AssertEquals_BOOL(TRUE, bResult, 'Failed to check if item is in map.');

	TEST_FINISHED();
END_METHOD

METHOD Check_If_Get_Key_Values_Returns_Keys_In_Specified_Order
VAR_INST
	fbMap : FB_Tree_Map;
	arnItems : ARRAY[0..3] OF DINT := [1,2,3,4];
	arnIn_Order, arnPre_Order, arnPost_Order, arnLevel_Order : ARRAY[0..3] OF DINT;
	i : DINT;
END_VAR
// Checked using: https://www.cs.usfca.edu/~galles/visualization/AVLtree.html
TcUnit.TEST('Check_If_Get_Key_Values_Returns_Keys_In_Specified_Order');

	FOR i := 0 TO 3 DO
    	fbMap.Insert(arnItems[i], arnItems[i]);
    	END_FOR
		
	fbMap._Traversal := T_BST_Traversal.In_Order;
	fbMap.Get_Keys()
		.Get(0, arnIn_Order[0])
		.Get(1, arnIn_Order[1]);
	fbMap.Get_Keys()
		.Get(2, arnIn_Order[2])
		.Get(3, arnIn_Order[3]);
	THIS^.AssertEquals_DINT(1, arnIn_Order[0],'Failed to get key with in-order traversal.');
	THIS^.AssertEquals_DINT(2, arnIn_Order[1],'Failed to get key with in-order traversal.');
	THIS^.AssertEquals_DINT(3, arnIn_Order[2],'Failed to get key with in-order traversal.');
	THIS^.AssertEquals_DINT(4, arnIn_Order[3],'Failed to get key with in-order traversal.');
	
	fbMap.Get_Values()
		.Get(0, arnIn_Order[0])
		.Get(1, arnIn_Order[1]);
	fbMap.Get_Values()
		.Get(2, arnIn_Order[2])
		.Get(3, arnIn_Order[3]);
	THIS^.AssertEquals_DINT(1, arnIn_Order[0],'Failed to get values with in-order traversal.');
	THIS^.AssertEquals_DINT(2, arnIn_Order[1],'Failed to get values with in-order traversal.');
	THIS^.AssertEquals_DINT(3, arnIn_Order[2],'Failed to get values with in-order traversal.');
	THIS^.AssertEquals_DINT(4, arnIn_Order[3],'Failed to get values with in-order traversal.');
	
	fbMap._Traversal := T_BST_Traversal.Pre_Order;
	fbMap.Get_Keys()
		.Get(0, arnPre_Order[0])
		.Get(1, arnPre_Order[1]);
	fbMap.Get_Keys()
		.Get(2, arnPre_Order[2])
		.Get(3, arnPre_Order[3]);
	THIS^.AssertEquals_DINT(2, arnPre_Order[0],'Failed to get key with pre-order traversal.');
	THIS^.AssertEquals_DINT(1, arnPre_Order[1],'Failed to get key with pre-order traversal.');
	THIS^.AssertEquals_DINT(3, arnPre_Order[2],'Failed to get key with pre-order traversal.');
	THIS^.AssertEquals_DINT(4, arnPre_Order[3],'Failed to get key with pre-order traversal.');
	fbMap.Get_Values()
		.Get(0, arnPre_Order[0])
		.Get(1, arnPre_Order[1]);
	fbMap.Get_Values()
		.Get(2, arnPre_Order[2])
		.Get(3, arnPre_Order[3]);
	THIS^.AssertEquals_DINT(2, arnPre_Order[0],'Failed to get value with pre-order traversal.');
	THIS^.AssertEquals_DINT(1, arnPre_Order[1],'Failed to get value with pre-order traversal.');
	THIS^.AssertEquals_DINT(3, arnPre_Order[2],'Failed to get value with pre-order traversal.');
	THIS^.AssertEquals_DINT(4, arnPre_Order[3],'Failed to get value with pre-order traversal.');
	
	fbMap._Traversal := T_BST_Traversal.Post_Order; 
	fbMap.Get_Keys()
		.Get(0, arnPost_Order[0])
		.Get(1, arnPost_Order[1]);
	fbMap.Get_Keys()
		.Get(2, arnPost_Order[2])
		.Get(3, arnPost_Order[3]);
	THIS^.AssertEquals_DINT(1, arnPost_Order[0],'Failed to get key with post-order traversal.');
	THIS^.AssertEquals_DINT(4, arnPost_Order[1],'Failed to get key with post-order traversal.');
	THIS^.AssertEquals_DINT(3, arnPost_Order[2],'Failed to get key with post-order traversal.');
	THIS^.AssertEquals_DINT(2, arnPost_Order[3],'Failed to get key with post-order traversal.');
	fbMap.Get_Values()
		.Get(0, arnPost_Order[0])
		.Get(1, arnPost_Order[1]);
	fbMap.Get_Values()
		.Get(2, arnPost_Order[2])
		.Get(3, arnPost_Order[3]);
	THIS^.AssertEquals_DINT(1, arnPost_Order[0],'Failed to get value with post-order traversal.');
	THIS^.AssertEquals_DINT(4, arnPost_Order[1],'Failed to get value with post-order traversal.');
	THIS^.AssertEquals_DINT(3, arnPost_Order[2],'Failed to get value with post-order traversal.');
	THIS^.AssertEquals_DINT(2, arnPost_Order[3],'Failed to get value with post-order traversal.');
	
	fbMap._Traversal := T_BST_Traversal.Level_Order; // will get the values in ascending order
	fbMap.Get_Keys()
		.Get(0, arnLevel_Order[0])
		.Get(1, arnLevel_Order[1]);
	fbMap.Get_Keys()
		.Get(2, arnLevel_Order[2])
		.Get(3, arnLevel_Order[3]);
	THIS^.AssertEquals_DINT(2, arnLevel_Order[0],'Failed to get item with level-order traversal.');
	THIS^.AssertEquals_DINT(1, arnLevel_Order[1],'Failed to get item with level-order traversal.');
	THIS^.AssertEquals_DINT(3, arnLevel_Order[2],'Failed to get item with level-order traversal.');
	THIS^.AssertEquals_DINT(4, arnLevel_Order[3],'Failed to get item with level-order traversal.');
	fbMap.Get_Values()
		.Get(0, arnLevel_Order[0])
		.Get(1, arnLevel_Order[1]);
	fbMap.Get_Values()
		.Get(2, arnLevel_Order[2])
		.Get(3, arnLevel_Order[3]);
	THIS^.AssertEquals_DINT(2, arnLevel_Order[0],'Failed to get value with level-order traversal.');
	THIS^.AssertEquals_DINT(1, arnLevel_Order[1],'Failed to get value with level-order traversal.');
	THIS^.AssertEquals_DINT(3, arnLevel_Order[2],'Failed to get value with level-order traversal.');
	THIS^.AssertEquals_DINT(4, arnLevel_Order[3],'Failed to get value with level-order traversal.');
	
	TEST_FINISHED();
END_METHOD

METHOD Check_If_Insert_Adds_Items
VAR_INST
	fbMap : FB_Tree_Map;
	sItem : STRING := 'I love cats';
	nItem : INT := 42;
END_VAR
TcUnit.TEST('Check_If_Insert_Adds_Items');

	fbMap
		.Insert(sItem, nItem)
		.Insert(nItem, sItem);
		
	THIS^.AssertEquals_DINT(2, fbMap._Count, 'Failed to insert items into map.');
	
	TEST_FINISHED();
END_METHOD

METHOD Check_If_Remove_Removes_Items
VAR_INST
	fbMap : FB_Tree_Map;
	sItem : STRING := 'I love cats';
	nItem : INT := 42;
	fItem : LREAL := 37.4;
END_VAR
TcUnit.TEST('Check_If_Remove_Removes_Items');

	fbMap
		.Insert(sItem, nItem)
		.Insert(nItem, fItem)
		.Insert(fItem, sItem)
		.Remove(nItem);
		
	THIS^.AssertEquals_DINT(2, fbMap._Count, 'Failed to remove item in set.');
	THIS^.AssertEquals_BOOL(TRUE, fbMap.Contains(sItem), 'Failed to remove item in set.');
	THIS^.AssertEquals_BOOL(FALSE, fbMap.Contains(nItem), 'Failed to remove item in set.');
	THIS^.AssertEquals_BOOL(TRUE, fbMap.Contains(fItem), 'Failed to remove item in set.');	
	
	TEST_FINISHED();
END_METHOD

METHOD Check_If_Update_Updates_Items
VAR_INST
	fbMap : FB_Tree_Map;
	sItem : STRING := 'I love cats';
	nItem : INT := 42;
	fItem : LREAL := 37.4;
	fNew_Item : LREAL := 3.14;
	fR_Item,
	fR_Updated_Item : LREAL;
END_VAR
TcUnit.TEST('Check_If_Update_Updates_Items');
	fbMap
		.Insert(sItem, nItem)
		.Insert(nItem, fItem)
		.Insert(fItem, sItem)
		.Get(nItem, fR_Item)
		.Update(nItem, fNew_Item)
		.Get(nItem, fR_Updated_Item);
	
	THIS^.AssertEquals_LREAL(37.4, fR_Item, 0.0001, 'Failed to get value to be updated in map.');
	THIS^.AssertEquals_LREAL(3.14, fR_Updated_Item, 0.0001, 'Failed to get updated value in map.');
		
	TEST_FINISHED();
END_METHOD

METHOD Check_If_Upsert_Updates_Items_Or_Adds_If_They_Dont_Exist
VAR_INST
	fbMap : FB_Tree_Map;
	nItem : INT := 42;
	fItem : LREAL := 37.4;
	fNew_Item : LREAL := 3.14;
	fR_Item,
	fR_Updated_Item : LREAL;
END_VAR
TcUnit.TEST('Check_If_Upsert_Updates_Items_Or_Adds_If_They_Dont_Exist');
	fbMap
		.Upsert(nItem, fItem)
		.Get(nItem, fR_Item)
		.Upsert(nItem, fNew_Item)
		.Get(nItem, fR_Updated_Item);
		
	THIS^.AssertEquals_LREAL(37.4, fR_Item, 0.0001, 'Failed to insert key value in map.');
	THIS^.AssertEquals_LREAL(3.14, fR_Updated_Item, 0.0001, 'Failed to update value in map.');
	TEST_FINISHED();
END_METHOD

END_FUNCTION_BLOCK

// ---- POUs/Function Blocks/FB_Tree_Multiset_Test_Suite.TcPOU
FUNCTION_BLOCK FB_Tree_Multiset_Test_Suite EXTENDS TcUnit.FB_TestSuite
VAR
END_VAR

Check_If_Clear_Empties_Items();
Check_If_Contains_Returns_True_If_Item_In_Set();
Check_If_Duplicate_Items_Can_Be_Inserted();
Check_If_Get_Values_Returns_Values_In_Specified_Order();
Check_If_Insert_Adds_Items();
Check_If_Remove_Removes_Items();
Check_If_Balanced_After_Removing_From_Left_Heavy_Tree();

METHOD Check_If_Balanced_After_Removing_From_Left_Heavy_Tree
VAR_INST
	fbSet : FB_Tree_Multiset;
	i, j : INT;
	arnItems : ARRAY[0..2] OF INT;
	ipItems : I_Immutable_List;
END_VAR
TcUnit.TEST('Check_If_Balanced_After_Removing_From_Left_Heavy_Tree');
	FOR i := 4 TO 1 BY -1 DO fbSet.Insert(i); END_FOR

	j := 3;
	fbSet._Traversal := T_BST_Traversal.Level_Order;
	ipItems := fbSet.Remove(j).Get_Values();

	ipItems
		.Get(0, arnItems[0])
		.Get(1, arnItems[1])
		.Get(2, arnItems[2]);
			
	THIS^.AssertEquals_DINT(3, fbSet._Count, 'Incorrect number of items retrieved after removing root item.');
	THIS^.AssertEquals_INT(2, arnItems[0], 'First value in level-order traversal is incorrect.');
	THIS^.AssertEquals_INT(1, arnItems[1], 'Second value in level-order traversal is incorrect.');
	THIS^.AssertEquals_INT(4, arnItems[2], 'Third value in level-order traversal is incorrect.');

TEST_FINISHED();
END_METHOD

METHOD Check_If_Clear_Empties_Items
VAR_INST
	fbSet : FB_Tree_Multiset;
	sItem : STRING := 'I love cats';
	nItem : INT := 42;
END_VAR
TcUnit.TEST('Check_If_Clear_Empties');
	fbSet
		.Insert(sItem)
		.Insert(nItem)
		.Clear();
		
	THIS^.AssertEquals_DINT(0, fbSet._Count, 'Set was not empty after inserting data.');
	
	TEST_FINISHED();
END_METHOD

METHOD Check_If_Contains_Returns_True_If_Item_In_Set
VAR_INST
	fbSet : FB_Tree_Multiset;
	sItem : STRING := 'I love cats';
	nItem : INT := 42;
	bResult : BOOL;
END_VAR
TcUnit.TEST('Check_If_Contains_Returns_True_If_Item_In_Set');

	bResult := fbSet
		.Insert(sItem)
		.Insert(nItem)
		.Contains(nItem);
		
	THIS^.AssertEquals_BOOL(TRUE, bResult, 'Failed to check if item is in set.');
	TEST_FINISHED();
END_METHOD

METHOD Check_If_Duplicate_Items_Can_Be_Inserted
VAR_INST
	fbSet : FB_Tree_Multiset;
	arnItems : ARRAY[0..5] OF DINT := [3,1,2,1,3,2];
	arnItems2 : ARRAY[0..5] OF DINT;
	ipItems : I_Immutable_List;
	i : DINT;
END_VAR
TcUnit.TEST('Check_If_Duplicate_Items_Can_Be_Inserted');

	FOR i := 0 TO 5 DO
    	fbSet.Insert(arnItems[i]);
    	END_FOR
		
	THIS^.AssertEquals_DINT(6, fbSet._Count, 'Multiset failed to insert duplicate items.');
	
	fbSet._Traversal := T_BST_Traversal.In_Order; // will get the values in ascending order

	ipItems := fbSet.Get_Values();
	ipItems
		.Get(0, arnItems2[0])
		.Get(1, arnItems2[1])
		.Get(2, arnItems2[2])
		.Get(3, arnItems2[3])
		.Get(4, arnItems2[4])
		.Get(5, arnItems2[5]);
		
	THIS^.AssertEquals_DINT(1, arnItems2[0],'');
	THIS^.AssertEquals_DINT(1, arnItems2[1],'');
	THIS^.AssertEquals_DINT(2, arnItems2[2],'');
	THIS^.AssertEquals_DINT(2, arnItems2[3],'');
	THIS^.AssertEquals_DINT(3, arnItems2[4],'');
	THIS^.AssertEquals_DINT(3, arnItems2[5],'');
		
	TEST_FINISHED();
END_METHOD

METHOD Check_If_Get_Values_Returns_Values_In_Specified_Order
VAR_INST
	fbSet : FB_Tree_Multiset;
	arnItems : ARRAY[0..3] OF DINT := [1,2,3,4];
	arnIn_Order, arnPre_Order, arnPost_Order, arnLevel_Order : ARRAY[0..3] OF DINT;
	ipItems : I_Immutable_List;
	i : DINT;
END_VAR
// Checked using: https://www.cs.usfca.edu/~galles/visualization/AVLtree.html
TcUnit.TEST('Check_If_Get_Values_Returns_Values_In_Specified_Order');

	FOR i := 0 TO 3 DO
    	fbSet.Insert(arnItems[i]);
    	END_FOR
		
	fbSet._Traversal := T_BST_Traversal.In_Order;
	ipItems := fbSet.Get_Values();
	ipItems
		.Get(0, arnIn_Order[0])
		.Get(1, arnIn_Order[1])
		.Get(2, arnIn_Order[2])
		.Get(3, arnIn_Order[3]);
	THIS^.AssertEquals_DINT(1, arnIn_Order[0],'Failed to get item with in-order traversal.');
	THIS^.AssertEquals_DINT(2, arnIn_Order[1],'Failed to get item with in-order traversal.');
	THIS^.AssertEquals_DINT(3, arnIn_Order[2],'Failed to get item with in-order traversal.');
	THIS^.AssertEquals_DINT(4, arnIn_Order[3],'Failed to get item with in-order traversal.');
	
	fbSet._Traversal := T_BST_Traversal.Pre_Order;
	ipItems := fbSet.Get_Values();
	ipItems
		.Get(0, arnPre_Order[0])
		.Get(1, arnPre_Order[1])
		.Get(2, arnPre_Order[2])
		.Get(3, arnPre_Order[3]);
	THIS^.AssertEquals_DINT(2, arnPre_Order[0],'Failed to get item with pre-order traversal.');
	THIS^.AssertEquals_DINT(1, arnPre_Order[1],'Failed to get item with pre-order traversal.');
	THIS^.AssertEquals_DINT(3, arnPre_Order[2],'Failed to get item with pre-order traversal.');
	THIS^.AssertEquals_DINT(4, arnPre_Order[3],'Failed to get item with pre-order traversal.');
	
	fbSet._Traversal := T_BST_Traversal.Post_Order; 
	ipItems := fbSet.Get_Values();
	ipItems
		.Get(0, arnPost_Order[0])
		.Get(1, arnPost_Order[1])
		.Get(2, arnPost_Order[2])
		.Get(3, arnPost_Order[3]);
	THIS^.AssertEquals_DINT(1, arnPost_Order[0],'Failed to get item with post-order traversal.');
	THIS^.AssertEquals_DINT(4, arnPost_Order[1],'Failed to get item with post-order traversal.');
	THIS^.AssertEquals_DINT(3, arnPost_Order[2],'Failed to get item with post-order traversal.');
	THIS^.AssertEquals_DINT(2, arnPost_Order[3],'Failed to get item with post-order traversal.');
	
	fbSet._Traversal := T_BST_Traversal.Level_Order; // will get the values in ascending order
	ipItems := fbSet.Get_Values();
	ipItems
		.Get(0, arnLevel_Order[0])
		.Get(1, arnLevel_Order[1])
		.Get(2, arnLevel_Order[2])
		.Get(3, arnLevel_Order[3]);
	THIS^.AssertEquals_DINT(2, arnLevel_Order[0],'Failed to get item with level-order traversal.');
	THIS^.AssertEquals_DINT(1, arnLevel_Order[1],'Failed to get item with level-order traversal.');
	THIS^.AssertEquals_DINT(3, arnLevel_Order[2],'Failed to get item with level-order traversal.');
	THIS^.AssertEquals_DINT(4, arnLevel_Order[3],'Failed to get item with level-order traversal.');
	
	TEST_FINISHED();
END_METHOD

METHOD Check_If_Insert_Adds_Items
VAR_INST
	fbSet : FB_Tree_Multiset;
	sItem : STRING := 'I love cats';
	nItem : INT := 42;
END_VAR
TcUnit.TEST('Check_If_Insert_Adds_Items');
	fbSet
		.Insert(sItem)
		.Insert(nItem);
		
	THIS^.AssertEquals_DINT(2, fbSet._Count, 'Failed to insert items into set.');
	
	TEST_FINISHED();
END_METHOD

METHOD Check_If_Remove_Removes_Items
VAR_INST
	fbSet : FB_Tree_Multiset;
	sItem : STRING := 'I love cats';
	nItem : INT := 42;
	fItem : LREAL := 37.4;
END_VAR
TcUnit.TEST('Check_If_Remove_Removes_Items');

	fbSet
		.Insert(sItem)
		.Insert(nItem)
		.Insert(fItem)
		.Remove(nItem);
		
	THIS^.AssertEquals_DINT(2, fbSet._Count, 'Failed to remove item in set.');
	THIS^.AssertEquals_BOOL(TRUE, fbSet.Contains(sItem), 'Failed to remove item in set.');
	THIS^.AssertEquals_BOOL(FALSE, fbSet.Contains(nItem), 'Failed to remove item in set.');
	THIS^.AssertEquals_BOOL(TRUE, fbSet.Contains(fItem), 'Failed to remove item in set.');	

	TEST_FINISHED();
END_METHOD

END_FUNCTION_BLOCK

// ---- POUs/Function Blocks/FB_Hash_Set_Test_Suite.TcPOU
FUNCTION_BLOCK FB_Hash_Set_Test_Suite EXTENDS TcUnit.FB_TestSuite
VAR
END_VAR

Check_If_Clear_Empties_Items();
Check_If_Contains_Returns_True_If_Item_In_Set();
Check_If_Duplicate_Items_Cannot_Be_Inserted();
Check_If_Get_Values_Returns_Values();
Check_If_Insert_Adds_Items();
Check_If_Remove_Removes_Items();

METHOD Check_If_Clear_Empties_Items
VAR_INST
	fbSet : FB_Hash_Set(0);
	sItem : STRING := 'I love cats';
	nItem : INT := 42;
END_VAR
TcUnit.TEST('Check_If_Clear_Empties');
	fbSet
		.Insert(sItem)
		.Insert(nItem)
		.Clear();
		
	THIS^.AssertEquals_DINT(0, fbSet._Count, 'Set was not empty after inserting data.');
	
	TEST_FINISHED();
END_METHOD

METHOD Check_If_Contains_Returns_True_If_Item_In_Set
VAR_INST
	fbSet : FB_Hash_Set(0);
	sItem : STRING := 'I love cats';
	nItem : INT := 42;
	bResult : BOOL;
END_VAR
TcUnit.TEST('Check_If_Contains_Returns_True_If_Item_In_Set');

	bResult := fbSet
		.Insert(sItem)
		.Insert(nItem)
		.Contains(nItem);
		
	THIS^.AssertEquals_BOOL(TRUE, bResult, 'Failed to check if item is in set.');
	TEST_FINISHED();
END_METHOD

METHOD Check_If_Duplicate_Items_Cannot_Be_Inserted
VAR_INST
	fbSet : FB_Hash_Set(0);
	arnItems : ARRAY[0..5] OF DINT := [3,1,2,1,3,2];
	i : DINT;
END_VAR
TcUnit.TEST('Check_If_Duplicate_Items_Cannot_Be_Inserted');

	FOR i := 0 TO 5 DO
    	fbSet.Insert(arnItems[i]);
    	END_FOR
		
	THIS^.AssertEquals_DINT(3, fbSet._Count, 'Set inserted duplicate items.');
		
	TEST_FINISHED();
END_METHOD

METHOD Check_If_Get_Values_Returns_Values
VAR_INST
	fbSet : FB_Hash_Set(0);
	arnItems : ARRAY[0..3] OF DINT := [1,2,3,4];
	arnReturned_Items : ARRAY[0..3] OF DINT;
	arIndex : ARRAY[0..3] OF T_Position := [4(-1)];
	i : DINT;
END_VAR
TcUnit.TEST('Check_If_Get_Values_Returns_Values');

	FOR i := 0 TO 3 DO
    	fbSet.Insert(arnItems[i]);
    	END_FOR
		
	fbSet.Get_Values()
		.Search(arnItems[0], index => arIndex[0])
		.Search(arnItems[1], index => arIndex[1])
		.Search(arnItems[2], index => arIndex[2])
		.Search(arnItems[3], index => arIndex[3]);
	fbSet.Get_Values()
		.Get(arIndex[0], arnReturned_Items[0])
		.Get(arIndex[1], arnReturned_Items[1])
		.Get(arIndex[2], arnReturned_Items[2])
		.Get(arIndex[3], arnReturned_Items[3]);
	THIS^.AssertEquals_DINT(1, arnReturned_Items[0],'');
	THIS^.AssertEquals_DINT(2, arnReturned_Items[1],'');
	THIS^.AssertEquals_DINT(3, arnReturned_Items[2],'');
	THIS^.AssertEquals_DINT(4, arnReturned_Items[3],'');
	
	TEST_FINISHED();
END_METHOD

METHOD Check_If_Insert_Adds_Items
VAR_INST
	fbSet : FB_Hash_Set(0);
	sItem : STRING := 'I love cats';
	nItem : INT := 42;
END_VAR
TcUnit.TEST('Check_If_Insert_Adds_Items');
	fbSet
		.Insert(sItem)
		.Insert(nItem);
		
	THIS^.AssertEquals_DINT(2, fbSet._Count, 'Failed to insert items into set.');
	
	TEST_FINISHED();
END_METHOD

METHOD Check_If_Remove_Removes_Items
VAR_INST
	fbSet : FB_Hash_Set(0);
	sItem : STRING := 'I love cats';
	nItem : INT := 42;
	fItem : LREAL := 37.4;
END_VAR
TcUnit.TEST('Check_If_Remove_Removes_Items');

	fbSet
		.Insert(sItem)
		.Insert(nItem)
		.Insert(fItem)
		.Remove(nItem);
		
	THIS^.AssertEquals_DINT(2, fbSet._Count, 'Failed to remove item in set.');
	THIS^.AssertEquals_BOOL(TRUE, fbSet.Contains(sItem), 'Failed to remove item in set.');
	THIS^.AssertEquals_BOOL(FALSE, fbSet.Contains(nItem), 'Failed to remove item in set.');
	THIS^.AssertEquals_BOOL(TRUE, fbSet.Contains(fItem), 'Failed to remove item in set.');	

	TEST_FINISHED();
END_METHOD

END_FUNCTION_BLOCK

// ---- POUs/Function Blocks/FB_Hash_Map_Test_Suite.TcPOU
FUNCTION_BLOCK FB_Hash_Map_Test_Suite EXTENDS TcUnit.FB_TestSuite
VAR
END_VAR

Check_If_Clear_Empties_Items();
Check_If_Insert_Adds_Items();
Check_If_Update_Updates_Items();
Check_If_Upsert_Updates_Items_Or_Adds_If_They_Dont_Exist();
Check_If_Remove_Removes_Items();
Check_If_Contains_Returns_True_If_Key_In_Map();
Check_If_Get_Key_Values_Returns_Keys_Values();

METHOD Check_If_Clear_Empties_Items
VAR_INST
	fbMap : FB_Hash_Map(0);
	sKey : STRING := 'I love cats';
	nValue : INT := 42;
END_VAR
TcUnit.TEST('Check_If_Clear_Empties');
	fbMap
		.Insert(sKey, nValue)
		.Clear();
		
	THIS^.AssertEquals_DINT(0, fbMap._Count, 'Map was not empty after inserting data.');
	
	TEST_FINISHED();
END_METHOD

METHOD Check_If_Contains_Returns_True_If_Key_In_Map
VAR_INST
	fbMap : FB_Hash_Map(0);
	sItem : STRING := 'I love cats';
	nItem : INT := 42;
	bResult : BOOL;
END_VAR
TcUnit.TEST('Check_If_Contains_Returns_True_If_Key_In_Map');

	bResult := fbMap
		.Insert(sItem, nItem)
		.Insert(nItem, sItem)
		.Contains(nItem);
		
	THIS^.AssertEquals_BOOL(TRUE, bResult, 'Failed to check if item is in map.');

	TEST_FINISHED();
END_METHOD

METHOD Check_If_Get_Key_Values_Returns_Keys_Values
VAR_INST
	fbMap : FB_Hash_Map(0);
	arnItems : ARRAY[0..3] OF DINT := [1,2,3,4];
	arnReturned_Keys,
	arnReturned_Values : ARRAY[0..3] OF DINT;
	arIndex : ARRAY[0..3] OF T_Position := [4(-1)];
	i : DINT;
END_VAR
TcUnit.TEST('Check_If_Get_Key_Values_Returns_Keys_Values');

	FOR i := 0 TO 3 DO
    	fbMap.Insert(arnItems[i], arnItems[i]);
    	END_FOR

	fbMap.Get_Keys()
		.Search(arnItems[0], index => arIndex[0])
		.Search(arnItems[1], index => arIndex[1])
		.Search(arnItems[2], index => arIndex[2])
		.Search(arnItems[3], index => arIndex[3]);
	fbMap.Get_Keys()
		.Get(arIndex[0], arnReturned_Keys[0])
		.Get(arIndex[1], arnReturned_Keys[1])
		.Get(arIndex[2], arnReturned_Keys[2])
		.Get(arIndex[3], arnReturned_Keys[3]);
	THIS^.AssertEquals_DINT(1, arnReturned_Keys[0],'');
	THIS^.AssertEquals_DINT(2, arnReturned_Keys[1],'');
	THIS^.AssertEquals_DINT(3, arnReturned_Keys[2],'');
	THIS^.AssertEquals_DINT(4, arnReturned_Keys[3],'');
	
	fbMap.Get_Values()
		.Get(arIndex[0], arnReturned_Values[0])
		.Get(arIndex[1], arnReturned_Values[1]);
	fbMap.Get_Values()
		.Get(arIndex[2], arnReturned_Values[2])
		.Get(arIndex[3], arnReturned_Values[3]);
	THIS^.AssertEquals_DINT(1, arnReturned_Values[0],'');
	THIS^.AssertEquals_DINT(2, arnReturned_Values[1],'');
	THIS^.AssertEquals_DINT(3, arnReturned_Values[2],'');
	THIS^.AssertEquals_DINT(4, arnReturned_Values[3],'');
	
	TEST_FINISHED();
END_METHOD

METHOD Check_If_Insert_Adds_Items
VAR_INST
	fbMap : FB_Hash_Map(0);
	sItem : STRING := 'I love cats';
	nItem : INT := 42;
END_VAR
TcUnit.TEST('Check_If_Insert_Adds_Items');

	fbMap
		.Insert(sItem, nItem)
		.Insert(nItem, sItem);
		
	THIS^.AssertEquals_DINT(2, fbMap._Count, 'Failed to insert items into map.');
	
	TEST_FINISHED();
END_METHOD

METHOD Check_If_Remove_Removes_Items
VAR_INST
	fbMap : FB_Hash_Map(0);
	sItem : STRING := 'I love cats';
	nItem : INT := 42;
	fItem : LREAL := 37.4;
END_VAR
TcUnit.TEST('Check_If_Remove_Removes_Items');

	fbMap
		.Insert(sItem, nItem)
		.Insert(nItem, fItem)
		.Insert(fItem, sItem)
		.Remove(nItem);
		
	THIS^.AssertEquals_DINT(2, fbMap._Count, 'Failed to remove item in set.');
	THIS^.AssertEquals_BOOL(TRUE, fbMap.Contains(sItem), 'Failed to remove item in set.');
	THIS^.AssertEquals_BOOL(FALSE, fbMap.Contains(nItem), 'Failed to remove item in set.');
	THIS^.AssertEquals_BOOL(TRUE, fbMap.Contains(fItem), 'Failed to remove item in set.');	
	
	TEST_FINISHED();
END_METHOD

METHOD Check_If_Update_Updates_Items
VAR_INST
	fbMap : FB_Hash_Map(0);
	sItem : STRING := 'I love cats';
	nItem : INT := 42;
	fItem : LREAL := 37.4;
	fNew_Item : LREAL := 3.14;
	fR_Item,
	fR_Updated_Item : LREAL;
END_VAR
TcUnit.TEST('Check_If_Update_Updates_Items');
	fbMap
		.Insert(sItem, nItem)
		.Insert(nItem, fItem)
		.Insert(fItem, sItem)
		.Get(nItem, fR_Item)
		.Update(nItem, fNew_Item)
		.Get(nItem, fR_Updated_Item);
	
	THIS^.AssertEquals_LREAL(37.4, fR_Item, 0.0001, 'Failed to get value to be updated in map.');
	THIS^.AssertEquals_LREAL(3.14, fR_Updated_Item, 0.0001, 'Failed to get updated value in map.');
		
	TEST_FINISHED();
END_METHOD

METHOD Check_If_Upsert_Updates_Items_Or_Adds_If_They_Dont_Exist
VAR_INST
	fbMap : FB_Hash_Map(0);
	nItem : INT := 42;
	fItem : LREAL := 37.4;
	fNew_Item : LREAL := 3.14;
	fR_Item,
	fR_Updated_Item : LREAL;
END_VAR
TcUnit.TEST('Check_If_Upsert_Updates_Items_Or_Adds_If_They_Dont_Exist');
	fbMap
		.Upsert(nItem, fItem)
		.Get(nItem, fR_Item)
		.Upsert(nItem, fNew_Item)
		.Get(nItem, fR_Updated_Item);
		
	THIS^.AssertEquals_LREAL(37.4, fR_Item, 0.0001, 'Failed to insert key value in map.');
	THIS^.AssertEquals_LREAL(3.14, fR_Updated_Item, 0.0001, 'Failed to update value in map.');
	TEST_FINISHED();
END_METHOD

END_FUNCTION_BLOCK

// ---- POUs/Function Blocks/FB_Ordered_Hash_Set_Test_Suite.TcPOU
FUNCTION_BLOCK FB_Ordered_Hash_Set_Test_Suite EXTENDS TcUnit.FB_TestSuite
VAR
END_VAR

Check_If_Clear_Empties_Items();
Check_If_Contains_Returns_True_If_Item_In_Set();
Check_If_Duplicate_Items_Cannot_Be_Inserted();
Check_If_Get_Values_Returns_Values();
Check_If_Insert_Adds_Items();
Check_If_Remove_Head_Item();
Check_If_Remove_Last_Remaining_Item();
Check_If_Remove_Removes_Items();

METHOD Check_If_Clear_Empties_Items
VAR_INST
	fbSet : FB_Ordered_Hash_Set(0);
	sItem : STRING := 'I love cats';
	nItem : INT := 42;
END_VAR
TcUnit.TEST('Check_If_Clear_Empties');
	fbSet
		.Insert(sItem)
		.Insert(nItem)
		.Clear();
		
	THIS^.AssertEquals_DINT(0, fbSet._Count, 'Set was not empty after inserting data.');
	
	TEST_FINISHED();
END_METHOD

METHOD Check_If_Contains_Returns_True_If_Item_In_Set
VAR_INST
	fbSet : FB_Ordered_Hash_Set(0);
	sItem : STRING := 'I love cats';
	nItem : INT := 42;
	bResult : BOOL;
END_VAR
TcUnit.TEST('Check_If_Contains_Returns_True_If_Item_In_Set');

	bResult := fbSet
		.Insert(sItem)
		.Insert(nItem)
		.Contains(nItem);
		
	THIS^.AssertEquals_BOOL(TRUE, bResult, 'Failed to check if item is in set.');
	TEST_FINISHED();
END_METHOD

METHOD Check_If_Duplicate_Items_Cannot_Be_Inserted
VAR_INST
	fbSet : FB_Ordered_Hash_Set(0);
	arnItems : ARRAY[0..5] OF DINT := [3,1,2,1,3,2];
	i : DINT;
END_VAR
TcUnit.TEST('Check_If_Duplicate_Items_Cannot_Be_Inserted');

	FOR i := 0 TO 5 DO
    	fbSet.Insert(arnItems[i]);
    	END_FOR
		
	THIS^.AssertEquals_DINT(3, fbSet._Count, 'Set inserted duplicate items.');
		
	TEST_FINISHED();
END_METHOD

METHOD Check_If_Get_Values_Returns_Values
VAR_INST
	fbSet : FB_Ordered_Hash_Set(0);
	arnItems : ARRAY[0..3] OF DINT := [1,2,3,4];
	arnReturned_Items : ARRAY[0..3] OF DINT;
	i : DINT;
END_VAR
TcUnit.TEST('Check_If_Get_Values_Returns_Values');

	FOR i := 0 TO 3 DO
    	fbSet.Insert(arnItems[i]);
    	END_FOR
		
	fbSet.Get_Values()
		.Get(0, arnReturned_Items[0])
		.Get(1, arnReturned_Items[1])
		.Get(2, arnReturned_Items[2])
		.Get(3, arnReturned_Items[3]);
		
	THIS^.AssertEquals_DINT(1, arnReturned_Items[0],'');
	THIS^.AssertEquals_DINT(2, arnReturned_Items[1],'');
	THIS^.AssertEquals_DINT(3, arnReturned_Items[2],'');
	THIS^.AssertEquals_DINT(4, arnReturned_Items[3],'');
	
	TEST_FINISHED();
END_METHOD

METHOD Check_If_Insert_Adds_Items
VAR_INST
	fbSet : FB_Ordered_Hash_Set(0);
	sItem : STRING := 'I love cats';
	nItem : INT := 42;
END_VAR
TcUnit.TEST('Check_If_Insert_Adds_Items');
	fbSet
		.Insert(sItem)
		.Insert(nItem);
		
	THIS^.AssertEquals_DINT(2, fbSet._Count, 'Failed to insert items into set.');
	
	TEST_FINISHED();
END_METHOD

METHOD Check_If_Remove_Head_Item : REFERENCE TO FB_Test
VAR_INST
	fbSet 		: FB_Ordered_Hash_Set(0);
	nFirst 		: INT := 1;
	nSecond 	: INT := 2;
	nThird 		: INT := 3;
	arnReturned : ARRAY[0..1] OF INT;
END_VAR
TcUnit.TEST('Check_If_Remove_Head_Item');

	fbSet
		.Insert(nFirst)
		.Insert(nSecond)
		.Insert(nThird)
		.Remove(nFirst);
	
	THIS^.AssertEquals_DINT(2, fbSet._Count, 'Count incorrect after removing head.');
	THIS^.AssertEquals_BOOL(FALSE, fbSet.Contains(nFirst), 'Head item still in set after removal.');
	
	fbSet.Get_Values()
		.Get(0, arnReturned[0])
		.Get(1, arnReturned[1]);
	
	THIS^.AssertEquals_DINT(2, arnReturned[0], 'Insertion order broken after head removal.');
	THIS^.AssertEquals_DINT(3, arnReturned[1], 'Insertion order broken after head removal.');
	
	TEST_FINISHED();
END_METHOD

METHOD Check_If_Remove_Last_Remaining_Item
VAR_INST
	fbSet : FB_Ordered_Hash_Set(0);
	nItem : INT := 42;
END_VAR
TcUnit.TEST('Check_If_Remove_Last_Remaining_Item');

	fbSet
		.Insert(nItem)
		.Remove(nItem);
	
	THIS^.AssertEquals_DINT(0, fbSet._Count, 'Failed to remove last remaining item.');
	THIS^.AssertEquals_BOOL(FALSE, fbSet.Contains(nItem), 'Set still contains item after removal.');
	
	TEST_FINISHED();
END_METHOD

METHOD Check_If_Remove_Removes_Items
VAR_INST
	fbSet : FB_Ordered_Hash_Set(0);
	sItem : STRING := 'I love cats';
	nItem : INT := 42;
	fItem : LREAL := 37.4;
END_VAR
TcUnit.TEST('Check_If_Remove_Removes_Items');

	fbSet
		.Insert(sItem)
		.Insert(nItem)
		.Insert(fItem)
		.Remove(nItem);
		
	THIS^.AssertEquals_DINT(2, fbSet._Count, 'Failed to remove item in set.');
	THIS^.AssertEquals_BOOL(TRUE, fbSet.Contains(sItem), 'Failed to remove item in set.');
	THIS^.AssertEquals_BOOL(FALSE, fbSet.Contains(nItem), 'Failed to remove item in set.');
	THIS^.AssertEquals_BOOL(TRUE, fbSet.Contains(fItem), 'Failed to remove item in set.');	

	TEST_FINISHED();
END_METHOD

END_FUNCTION_BLOCK

// ---- POUs/Function Blocks/FB_Ordered_Hash_Map_Test_Suite.TcPOU
FUNCTION_BLOCK FB_Ordered_Hash_Map_Test_Suite EXTENDS TcUnit.FB_TestSuite
VAR
END_VAR

Check_If_Clear_Empties_Items();
Check_If_Insert_Adds_Items();
Check_If_Update_Updates_Items();
Check_If_Upsert_Updates_Items_Or_Adds_If_They_Dont_Exist();
Check_If_Remove_Removes_Items();
Check_If_Contains_Returns_True_If_Key_In_Map();
Check_If_Get_Key_Values_Returns_Keys_Values();

METHOD Check_If_Clear_Empties_Items
VAR_INST
	fbMap : FB_Ordered_Hash_Map(0);
	sKey : STRING := 'I love cats';
	nValue : INT := 42;
END_VAR
TcUnit.TEST('Check_If_Clear_Empties');
	fbMap
		.Insert(sKey, nValue)
		.Clear();
		
	THIS^.AssertEquals_DINT(0, fbMap._Count, 'Map was not empty after inserting data.');
	
	TEST_FINISHED();
END_METHOD

METHOD Check_If_Contains_Returns_True_If_Key_In_Map
VAR_INST
	fbMap : FB_Ordered_Hash_Map(0);
	sItem : STRING := 'I love cats';
	nItem : INT := 42;
	bResult : BOOL;
END_VAR
TcUnit.TEST('Check_If_Contains_Returns_True_If_Key_In_Map');

	bResult := fbMap
		.Insert(sItem, nItem)
		.Insert(nItem, sItem)
		.Contains(nItem);
		
	THIS^.AssertEquals_BOOL(TRUE, bResult, 'Failed to check if item is in map.');

	TEST_FINISHED();
END_METHOD

METHOD Check_If_Get_Key_Values_Returns_Keys_Values
VAR_INST
	fbMap : FB_Ordered_Hash_Map(0);
	arnItems : ARRAY[0..3] OF DINT := [1,2,3,4];
	arnReturned_Keys,
	arnReturned_Values : ARRAY[0..3] OF DINT;
	i : DINT;
END_VAR
TcUnit.TEST('Check_If_Get_Key_Values_Returns_Keys_Values');

	FOR i := 0 TO 3 DO
    	fbMap.Insert(arnItems[i], arnItems[i]);
    	END_FOR
		
	fbMap.Get_Keys()
		.Get(0, arnReturned_Keys[0])
		.Get(1, arnReturned_Keys[1]);
	fbMap.Get_Keys()
		.Get(2, arnReturned_Keys[2])
		.Get(3, arnReturned_Keys[3]);
	THIS^.AssertEquals_DINT(1, arnReturned_Keys[0],'');
	THIS^.AssertEquals_DINT(2, arnReturned_Keys[1],'');
	THIS^.AssertEquals_DINT(3, arnReturned_Keys[2],'');
	THIS^.AssertEquals_DINT(4, arnReturned_Keys[3],'');
	
	fbMap.Get_Values()
		.Get(0, arnReturned_Values[0])
		.Get(1, arnReturned_Values[1]);
	fbMap.Get_Values()
		.Get(2, arnReturned_Values[2])
		.Get(3, arnReturned_Values[3]);
	THIS^.AssertEquals_DINT(1, arnReturned_Values[0],'');
	THIS^.AssertEquals_DINT(2, arnReturned_Values[1],'');
	THIS^.AssertEquals_DINT(3, arnReturned_Values[2],'');
	THIS^.AssertEquals_DINT(4, arnReturned_Values[3],'');
	
	TEST_FINISHED();
END_METHOD

METHOD Check_If_Insert_Adds_Items
VAR_INST
	fbMap : FB_Ordered_Hash_Map(0);
	sItem : STRING := 'I love cats';
	nItem : INT := 42;
END_VAR
TcUnit.TEST('Check_If_Insert_Adds_Items');

	fbMap
		.Insert(sItem, nItem)
		.Insert(nItem, sItem);
		
	THIS^.AssertEquals_DINT(2, fbMap._Count, 'Failed to insert items into map.');
	
	TEST_FINISHED();
END_METHOD

METHOD Check_If_Remove_Removes_Items
VAR_INST
	fbMap : FB_Ordered_Hash_Map(0);
	sItem : STRING := 'I love cats';
	nItem : INT := 42;
	fItem : LREAL := 37.4;
END_VAR
TcUnit.TEST('Check_If_Remove_Removes_Items');

	fbMap
		.Insert(sItem, nItem)
		.Insert(nItem, fItem)
		.Insert(fItem, sItem)
		.Remove(nItem);
		
	THIS^.AssertEquals_DINT(2, fbMap._Count, 'Failed to remove item in set.');
	THIS^.AssertEquals_BOOL(TRUE, fbMap.Contains(sItem), 'Failed to remove item in set.');
	THIS^.AssertEquals_BOOL(FALSE, fbMap.Contains(nItem), 'Failed to remove item in set.');
	THIS^.AssertEquals_BOOL(TRUE, fbMap.Contains(fItem), 'Failed to remove item in set.');	
	
	TEST_FINISHED();
END_METHOD

METHOD Check_If_Update_Updates_Items
VAR_INST
	fbMap : FB_Ordered_Hash_Map(0);
	sItem : STRING := 'I love cats';
	nItem : INT := 42;
	fItem : LREAL := 37.4;
	fNew_Item : LREAL := 3.14;
	fR_Item,
	fR_Updated_Item : LREAL;
END_VAR
TcUnit.TEST('Check_If_Update_Updates_Items');
	fbMap
		.Insert(sItem, nItem)
		.Insert(nItem, fItem)
		.Insert(fItem, sItem)
		.Get(nItem, fR_Item)
		.Update(nItem, fNew_Item)
		.Get(nItem, fR_Updated_Item);
	
	THIS^.AssertEquals_LREAL(37.4, fR_Item, 0.0001, 'Failed to get value to be updated in map.');
	THIS^.AssertEquals_LREAL(3.14, fR_Updated_Item, 0.0001, 'Failed to get updated value in map.');
		
	TEST_FINISHED();
END_METHOD

METHOD Check_If_Upsert_Updates_Items_Or_Adds_If_They_Dont_Exist
VAR_INST
	fbMap : FB_Ordered_Hash_Map(0);
	nItem : INT := 42;
	fItem : LREAL := 37.4;
	fNew_Item : LREAL := 3.14;
	fR_Item,
	fR_Updated_Item : LREAL;
END_VAR
TcUnit.TEST('Check_If_Upsert_Updates_Items_Or_Adds_If_They_Dont_Exist');
	fbMap
		.Upsert(nItem, fItem)
		.Get(nItem, fR_Item)
		.Upsert(nItem, fNew_Item)
		.Get(nItem, fR_Updated_Item);
		
	THIS^.AssertEquals_LREAL(37.4, fR_Item, 0.0001, 'Failed to insert key value in map.');
	THIS^.AssertEquals_LREAL(3.14, fR_Updated_Item, 0.0001, 'Failed to update value in map.');
	TEST_FINISHED();
END_METHOD

END_FUNCTION_BLOCK
